KUKA KRL program: EPS_2_25252_DC1_A_20250910061712.src

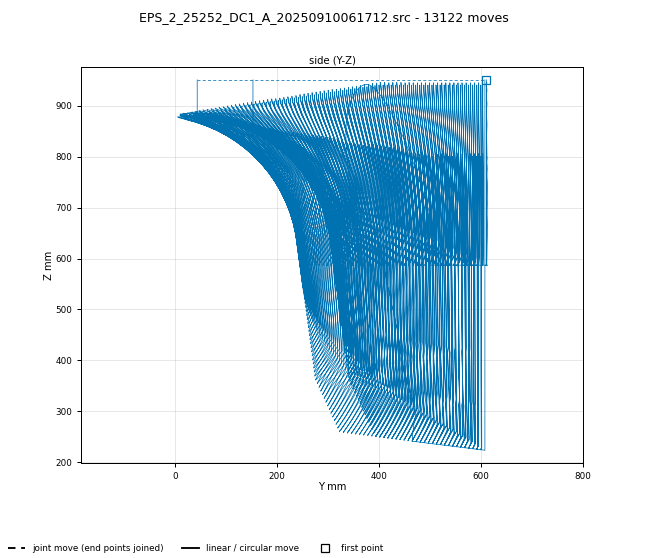
[picture p0: tool path of EPS_2_25252_DC1_A_20250910061712.src, 13122 of 13124 moves have a stored position in this frame; points joined in program order, loops and branches not executed]
&ACCESS RVP
&REL 4
&COMMENT QRS 19112012
&PARAM EDITMASK = *
DEF PART()
EXT BAS (BAS_COMMAND :IN,REAL :IN )
INT I
BAS (#INITMOV,0 )

;KUKA QRS Post kuka4.cps  Date:22-06-2017 !

File_ID=2828

QRS_PRE_INIT()

;Init var - Until changes are made in qrs_pre_init
Outlet_Square_prg=0
Inlet_1_Square_prg=0
Inlet_2_Square_prg=0
Inlet_3_Square_prg=0
Inlet_4_Square_prg=0
Inlet_5_Square_prg=0

Outlet_1={X 0.000, Y 400.000, Z 636.000, B 0.000, E1 0.000 }
Inlet_1={X 0.000, Y 504.550, Z 618.000, B 0.000, E1 206.000 }
Outlet_1_type=610
Inlet_1_type=366
;QRS#1=Sidecore dimensions
;QRS#2=600-24" Concrete
;QRS#3=375-15" PVC SDR 35
;QRS#4=
;QRS#5=
;QRS#6=
;QRS#7=
;QRS#8=
;QRS#9=S306-34L
;QRS#10=20Y PSX
;QRS#11=
;QRS#12=
;QRS#13=
;QRS#14=
;QRS#15=
;QRS#16=1220x127x1295 4,25'
;QRS#17=EPS Height
;QRS#18=941
;QRS#19=*
;QRS#20= UPDATED VERSION 22-06-2017
;QRS#21=*
Outlet_Square=0450
Inlet_1_Square=0250
Inlet_2_Square=0
Inlet_3_Square=0
Inlet_4_Square=0
Inlet_5_Square=0
Mill_Square=1
Outlet_Square_Prg=264
Inlet_1_Square_prg=252

QRS_INIT()

$ADVANCE=5

; T1
PTP {E1 178.399,E2 178.399}
PTP {X 0,Y 610.766,A -85,B 0,C 180,E1 178.399,E2 178.399,E3 0,E4 0,E5 0,E6 0}
QRS_SPEED_INIT()
LIN {X 0,Y 610.766,Z 951,A -85,B 0,C 180,E1 178.399,E2 178.399,E3 0,E4 0,E5 0,E6 0} C_VEL
LIN {X 0,Y 610.766,Z 588.94,A -85,B 0,C 180,E1 178.399,E2 178.399} C_VEL
LIN {X 0,Y 610.795,Z 586.94,A -85,B 0,C 180,E1 178.587,E2 178.587} C_VEL
LIN {X 0,Y 611.848,Z 586.94,A -85,B 0,C 180,E1 181.168,E2 181.168} C_VEL
LIN {X 0,Y 611.871,Z 586.94,A -85,B 0,C 180,E1 188.197,E2 188.197} C_VEL
LIN {X 0,Y 611.797,Z 586.94,A -85,B 0,C 180,E1 195.355,E2 195.355} C_VEL
LIN {X 0,Y 611.804,Z 586.94,A -85,B 0,C 180,E1 202.768,E2 202.768} C_VEL
LIN {X 0,Y 611.794,Z 586.94,A -85,B 0,C 180,E1 210.612,E2 210.612} C_VEL
LIN {X 0,Y 610.594,Z 586.94,A -85,B 0,C 180,E1 217.256,E2 217.256} C_VEL
LIN {X 0,Y 611.723,Z 586.94,A -85,B 0,C 180,E1 219.161,E2 219.161} C_VEL
LIN {X 0,Y 610.308,Z 586.94,A -85,B 0,C 180,E1 222.361,E2 222.361} C_VEL
LIN {X 0,Y 610.612,Z 586.94,A -85,B 0,C 180,E1 225.585,E2 225.585} C_VEL
LIN {X 0,Y 611.691,Z 586.94,A -85,B 0,C 180,E1 227.756,E2 227.756} C_VEL
LIN {X 0,Y 611.857,Z 586.94,A -85,B 0,C 180,E1 235.863,E2 235.863} C_VEL
LIN {X 0,Y 611.311,Z 586.94,A -85,B 0,C 180,E1 236.023,E2 236.023} C_VEL
LIN {X 0,Y 610.597,Z 586.94,A -85,B 0,C 180,E1 236.106,E2 236.106} C_VEL
LIN {X 0,Y 611.51,Z 647.546,A -85,B 0,C 180,E1 237.003,E2 237.003} C_VEL
LIN {X 0,Y 611.588,Z 668.499,A -85,B 0,C 180,E1 237.345,E2 237.345} C_VEL
LIN {X 0,Y 611.321,Z 684.266,A -85,B 0,C 180,E1 237.679,E2 237.679} C_VEL
LIN {X 0,Y 611.684,Z 698.104,A -85,B 0,C 180,E1 238.076,E2 238.076} C_VEL
LIN {X 0,Y 611.753,Z 713.122,A -85,B 0,C 180,E1 238.567,E2 238.567} C_VEL
LIN {X 0,Y 611.745,Z 728.257,A -85,B 0,C 180,E1 239.142,E2 239.142} C_VEL
LIN {X 0,Y 611.602,Z 742.813,A -85,B 0,C 180,E1 239.768,E2 239.768} C_VEL
LIN {X 0,Y 611.469,Z 748.567,A -85,B 0,C 180,E1 240.04,E2 240.04} C_VEL
LIN {X 0,Y 611.62,Z 757.431,A -85,B 0,C 180,E1 240.492,E2 240.492} C_VEL
LIN {X 0,Y 611.575,Z 770.08,A -85,B 0,C 180,E1 241.183,E2 241.183} C_VEL
LIN {X 0,Y 611.546,Z 782.628,A -85,B 0,C 180,E1 241.939,E2 241.939} C_VEL
LIN {X 0,Y 611.656,Z 796.717,A -85,B 0,C 180,E1 242.887,E2 242.887} C_VEL
LIN {X 0,Y 611.627,Z 808.354,A -85,B 0,C 180,E1 243.735,E2 243.735} C_VEL
LIN {X 0,Y 611.516,Z 820.103,A -85,B 0,C 180,E1 244.663,E2 244.663} C_VEL
LIN {X 0,Y 611.31,Z 832.04,A -85,B 0,C 180,E1 245.688,E2 245.688} C_VEL
LIN {X 0,Y 611.351,Z 842.488,A -85,B 0,C 180,E1 246.67,E2 246.67} C_VEL
LIN {X 0,Y 611.614,Z 852.795,A -85,B 0,C 180,E1 247.727,E2 247.727} C_VEL
LIN {X 0,Y 611.705,Z 861.779,A -85,B 0,C 180,E1 248.711,E2 248.711} C_VEL
LIN {X 0,Y 611.244,Z 871.74,A -85,B 0,C 180,E1 249.877,E2 249.877} C_VEL
LIN {X 0,Y 610.937,Z 881.3,A -85,B 0,C 180,E1 251.106,E2 251.106} C_VEL
LIN {X 0,Y 611.042,Z 888.988,A -85,B 0,C 180,E1 252.187,E2 252.187} C_VEL
LIN {X 0,Y 611.571,Z 897.667,A -85,B 0,C 180,E1 253.54,E2 253.54} C_VEL
LIN {X 0,Y 611.79,Z 901.959,A -85,B 0,C 180,E1 254.266,E2 254.266} C_VEL
LIN {X 0,Y 611.426,Z 906.652,A -85,B 0,C 180,E1 255.084,E2 255.084} C_VEL
LIN {X 0,Y 610.99,Z 912.543,A -85,B 0,C 180,E1 256.19,E2 256.19} C_VEL
LIN {X 0,Y 610.849,Z 918.046,A -85,B 0,C 180,E1 257.331,E2 257.331} C_VEL
LIN {X 0,Y 611.295,Z 924.36,A -85,B 0,C 180,E1 258.833,E2 258.833} C_VEL
LIN {X 0,Y 611.852,Z 928.798,A -85,B 0,C 180,E1 260.03,E2 260.03} C_VEL
LIN {X 0,Y 611.223,Z 932.641,A -85,B 0,C 180,E1 261.204,E2 261.204} C_VEL
LIN {X 0,Y 610.765,Z 935.979,A -85,B 0,C 180,E1 262.378,E2 262.378} C_VEL
LIN {X 0,Y 610.652,Z 937.542,A -85,B 0,C 180,E1 262.966,E2 262.966} C_VEL
LIN {X 0,Y 610.835,Z 940.117,A -85,B 0,C 180,E1 264.145,E2 264.145} C_VEL
LIN {X 0,Y 611.39,Z 942.182,A -85,B 0,C 180,E1 265.323,E2 265.323} C_VEL
LIN {X 0,Y 611.706,Z 943.787,A -85,B 0,C 180,E1 266.495,E2 266.495} C_VEL
LIN {X 0,Y 610.903,Z 945.157,A -85,B 0,C 180,E1 267.895,E2 267.895} C_VEL
LIN {X 0,Y 610.566,Z 945.724,A -85,B 0,C 180,E1 268.829,E2 268.829} C_VEL
LIN {X 0,Y 610.611,Z 945.959,A -85,B 0,C 180,E1 270.175,E2 270.175} C_VEL
LIN {X 0,Y 611.002,Z 945.713,A -85,B 0,C 180,E1 271.168,E2 271.168} C_VEL
LIN {X 0,Y 611.64,Z 945.019,A -85,B 0,C 180,E1 272.253,E2 272.253} C_VEL
LIN {X 0,Y 611.557,Z 944.17,A -85,B 0,C 180,E1 273.193,E2 273.193} C_VEL
LIN {X 0,Y 610.851,Z 942.2,A -85,B 0,C 180,E1 274.679,E2 274.679} C_VEL
LIN {X 0,Y 610.654,Z 940.123,A -85,B 0,C 180,E1 275.855,E2 275.855} C_VEL
LIN {X 0,Y 610.92,Z 937.546,A -85,B 0,C 180,E1 277.029,E2 277.029} C_VEL
LIN {X 0,Y 611.534,Z 934.39,A -85,B 0,C 180,E1 278.199,E2 278.199} C_VEL
LIN {X 0,Y 611.853,Z 932.642,A -85,B 0,C 180,E1 278.785,E2 278.785} C_VEL
LIN {X 0,Y 611.268,Z 928.807,A -85,B 0,C 180,E1 279.977,E2 279.977} C_VEL
LIN {X 0,Y 610.798,Z 923.162,A -85,B 0,C 180,E1 281.472,E2 281.472} C_VEL
LIN {X 0,Y 610.882,Z 918.056,A -85,B 0,C 180,E1 282.666,E2 282.666} C_VEL
LIN {X 0,Y 611.577,Z 910.301,A -85,B 0,C 180,E1 284.234,E2 284.234} C_VEL
LIN {X 0,Y 611.794,Z 906.723,A -85,B 0,C 180,E1 284.894,E2 284.894} C_VEL
LIN {X 0,Y 611.436,Z 902.319,A -85,B 0,C 180,E1 285.683,E2 285.683} C_VEL
LIN {X 0,Y 611.057,Z 897.089,A -85,B 0,C 180,E1 286.572,E2 286.572} C_VEL
LIN {X 0,Y 610.862,Z 887.941,A -85,B 0,C 180,E1 287.97,E2 287.97} C_VEL
LIN {X 0,Y 611.214,Z 879.031,A -85,B 0,C 180,E1 289.192,E2 289.192} C_VEL
LIN {X 0,Y 611.72,Z 869.206,A -85,B 0,C 180,E1 290.415,E2 290.415} C_VEL
LIN {X 0,Y 611.518,Z 859.844,A -85,B 0,C 180,E1 291.512,E2 291.512} C_VEL
LIN {X 0,Y 611.23,Z 849.887,A -85,B 0,C 180,E1 292.592,E2 292.592} C_VEL
LIN {X 0,Y 611.217,Z 839.652,A -85,B 0,C 180,E1 293.61,E2 293.61} C_VEL
LIN {X 0,Y 611.473,Z 828.289,A -85,B 0,C 180,E1 294.639,E2 294.639} C_VEL
LIN {X 0,Y 611.646,Z 817.642,A -85,B 0,C 180,E1 295.534,E2 295.534} C_VEL
LIN {X 0,Y 611.637,Z 805.784,A -85,B 0,C 180,E1 296.46,E2 296.46} C_VEL
LIN {X 0,Y 611.539,Z 793.169,A -85,B 0,C 180,E1 297.366,E2 297.366} C_VEL
LIN {X 0,Y 611.545,Z 780.808,A -85,B 0,C 180,E1 298.176,E2 298.176} C_VEL
LIN {X 0,Y 611.615,Z 766.332,A -85,B 0,C 180,E1 299.027,E2 299.027} C_VEL
LIN {X 0,Y 611.558,Z 756.226,A -85,B 0,C 180,E1 299.577,E2 299.577} C_VEL
LIN {X 0,Y 611.728,Z 739.176,A -85,B 0,C 180,E1 300.392,E2 300.392} C_VEL
LIN {X 0,Y 611.714,Z 723.993,A -85,B 0,C 180,E1 301.03,E2 301.03} C_VEL
LIN {X 0,Y 611.675,Z 709.715,A -85,B 0,C 180,E1 301.554,E2 301.554} C_VEL
LIN {X 0,Y 611.325,Z 695.349,A -85,B 0,C 180,E1 302.025,E2 302.025} C_VEL
LIN {X 0,Y 611.698,Z 679.814,A -85,B 0,C 180,E1 302.406,E2 302.406} C_VEL
LIN {X 0,Y 611.757,Z 665.783,A -85,B 0,C 180,E1 302.698,E2 302.698} C_VEL
LIN {X 0,Y 611.651,Z 645.532,A -85,B 0,C 180,E1 303.016,E2 303.016} C_VEL
LIN {X 0,Y 610.854,Z 596.983,A -85,B 0,C 180,E1 303.735,E2 303.735} C_VEL
LIN {X 0,Y 610.662,Z 586.94,A -85,B 0,C 180,E1 303.893,E2 303.893} C_VEL
LIN {X 0,Y 611.322,Z 586.94,A -85,B 0,C 180,E1 303.972,E2 303.972} C_VEL
LIN {X 0,Y 611.676,Z 586.94,A -85,B 0,C 180,E1 304.64,E2 304.64} C_VEL
LIN {X 0,Y 611.825,Z 586.94,A -85,B 0,C 180,E1 309.151,E2 309.151} C_VEL
LIN {X 0,Y 610.37,Z 586.94,A -85,B 0,C 180,E1 312.353,E2 312.353} C_VEL
LIN {X 0,Y 610.667,Z 586.94,A -85,B 0,C 180,E1 315.577,E2 315.577} C_VEL
LIN {X 0,Y 611.742,Z 586.94,A -85,B 0,C 180,E1 317.761,E2 317.761} C_VEL
LIN {X 0,Y 610.224,Z 586.94,A -85,B 0,C 180,E1 323.686,E2 323.686} C_VEL
LIN {X 0,Y 611.725,Z 586.94,A -85,B 0,C 180,E1 326.634,E2 326.634} C_VEL
LIN {X 0,Y 611.738,Z 586.94,A -85,B 0,C 180,E1 334.673,E2 334.673} C_VEL
LIN {X 0,Y 611.49,Z 586.94,A -85,B 0,C 180,E1 343.289,E2 343.289} C_VEL
LIN {X 0,Y 611.249,Z 586.94,A -85,B 0,C 180,E1 344.631,E2 344.631} C_VEL
LIN {X 0,Y 611.788,Z 586.94,A -85,B 0,C 180,E1 351.802,E2 351.802} C_VEL
LIN {X 0,Y 611.834,Z 586.94,A -85,B 0,C 180,E1 358.832,E2 358.832} C_VEL
LIN {X 0,Y 611.791,Z 586.94,A -85,B 0,C 180,E1 365.845,E2 365.845} C_VEL
LIN {X 0,Y 611.835,Z 586.94,A -85,B 0,C 180,E1 372.946,E2 372.946} C_VEL
LIN {X 0,Y 611.779,Z 586.94,A -85,B 0,C 180,E1 380.259,E2 380.259} C_VEL
LIN {X 0,Y 611.755,Z 586.94,A -85,B 0,C 180,E1 387.936,E2 387.936} C_VEL
LIN {X 0,Y 610.34,Z 586.94,A -85,B 0,C 180,E1 393.168,E2 393.168} C_VEL
LIN {X 0,Y 611.785,Z 586.94,A -85,B 0,C 180,E1 396.205,E2 396.205} C_VEL
LIN {X 0,Y 611.323,Z 586.94,A -85,B 0,C 180,E1 397.349,E2 397.349} C_VEL
LIN {X 0,Y 611.836,Z 586.94,A -85,B 0,C 180,E1 403.144,E2 403.144} C_VEL
LIN {X 0,Y 611.437,Z 586.94,A -85,B 0,C 180,E1 403.288,E2 403.288} C_VEL
LIN {X 0,Y 611.426,Z 596.264,A -85,B 0,C 180,E1 403.448,E2 403.448} C_VEL
LIN {X 0,Y 611.785,Z 623.475,A -85,B 0,C 180,E1 403.804,E2 403.804} C_VEL
LIN {X 0,Y 611.801,Z 632.118,A -85,B 0,C 180,E1 403.947,E2 403.947} C_VEL
LIN {X 0,Y 611.734,Z 641.309,A -85,B 0,C 180,E1 404.136,E2 404.136} C_VEL
LIN {X 0,Y 611.726,Z 648.588,A -85,B 0,C 180,E1 404.316,E2 404.316} C_VEL
LIN {X 0,Y 611.81,Z 658.939,A -85,B 0,C 180,E1 404.626,E2 404.626} C_VEL
LIN {X 0,Y 611.799,Z 668.311,A -85,B 0,C 180,E1 404.953,E2 404.953} C_VEL
LIN {X 0,Y 611.811,Z 677.548,A -85,B 0,C 180,E1 405.323,E2 405.323} C_VEL
LIN {X 0,Y 611.792,Z 686.258,A -85,B 0,C 180,E1 405.718,E2 405.718} C_VEL
LIN {X 0,Y 611.755,Z 693.578,A -85,B 0,C 180,E1 406.083,E2 406.083} C_VEL
LIN {X 0,Y 611.679,Z 703.091,A -85,B 0,C 180,E1 406.614,E2 406.614} C_VEL
LIN {X 0,Y 611.54,Z 712.053,A -85,B 0,C 180,E1 407.172,E2 407.172} C_VEL
LIN {X 0,Y 611.518,Z 719.064,A -85,B 0,C 180,E1 407.653,E2 407.653} C_VEL
LIN {X 0,Y 611.656,Z 726.904,A -85,B 0,C 180,E1 408.246,E2 408.246} C_VEL
LIN {X 0,Y 611.808,Z 734.808,A -85,B 0,C 180,E1 408.903,E2 408.903} C_VEL
LIN {X 0,Y 611.752,Z 740.864,A -85,B 0,C 180,E1 409.445,E2 409.445} C_VEL
LIN {X 0,Y 611.519,Z 747.37,A -85,B 0,C 180,E1 410.073,E2 410.073} C_VEL
LIN {X 0,Y 611.286,Z 754.307,A -85,B 0,C 180,E1 410.808,E2 410.808} C_VEL
LIN {X 0,Y 611.275,Z 759.983,A -85,B 0,C 180,E1 411.467,E2 411.467} C_VEL
LIN {X 0,Y 611.474,Z 765.259,A -85,B 0,C 180,E1 412.136,E2 412.136} C_VEL
LIN {X 0,Y 611.815,Z 771.733,A -85,B 0,C 180,E1 413.047,E2 413.047} C_VEL
LIN {X 0,Y 611.775,Z 774.744,A -85,B 0,C 180,E1 413.495,E2 413.495} C_VEL
LIN {X 0,Y 611.312,Z 780.353,A -85,B 0,C 180,E1 414.417,E2 414.417} C_VEL
LIN {X 0,Y 611.03,Z 784.515,A -85,B 0,C 180,E1 415.18,E2 415.18} C_VEL
LIN {X 0,Y 611.072,Z 789.541,A -85,B 0,C 180,E1 416.243,E2 416.243} C_VEL
LIN {X 0,Y 611.399,Z 792.933,A -85,B 0,C 180,E1 417.064,E2 417.064} C_VEL
LIN {X 0,Y 611.88,Z 796.656,A -85,B 0,C 180,E1 418.124,E2 418.124} C_VEL
LIN {X 0,Y 611.543,Z 798.59,A -85,B 0,C 180,E1 418.743,E2 418.743} C_VEL
LIN {X 0,Y 611.002,Z 801.321,A -85,B 0,C 180,E1 419.81,E2 419.81} C_VEL
LIN {X 0,Y 610.85,Z 802.311,A -85,B 0,C 180,E1 420.263,E2 420.263} C_VEL
LIN {X 0,Y 610.888,Z 804.098,A -85,B 0,C 180,E1 421.298,E2 421.298} C_VEL
LIN {X 0,Y 611.19,Z 804.968,A -85,B 0,C 180,E1 422.036,E2 422.036} C_VEL
LIN {X 0,Y 611.725,Z 805.707,A -85,B 0,C 180,E1 423.014,E2 423.014} C_VEL
LIN {X 0,Y 611.599,Z 805.938,A -85,B 0,C 180,E1 423.841,E2 423.841} C_VEL
LIN {X 0,Y 611.17,Z 805.82,A -85,B 0,C 180,E1 424.65,E2 424.65} C_VEL
LIN {X 0,Y 610.885,Z 805.27,A -85,B 0,C 180,E1 425.565,E2 425.565} C_VEL
LIN {X 0,Y 610.97,Z 804.103,A -85,B 0,C 180,E1 426.607,E2 426.607} C_VEL
LIN {X 0,Y 611.606,Z 801.736,A -85,B 0,C 180,E1 427.897,E2 427.897} C_VEL
LIN {X 0,Y 611.834,Z 800.373,A -85,B 0,C 180,E1 428.496,E2 428.496} C_VEL
LIN {X 0,Y 611.547,Z 798.741,A -85,B 0,C 180,E1 429.111,E2 429.111} C_VEL
LIN {X 0,Y 611.047,Z 794.846,A -85,B 0,C 180,E1 430.338,E2 430.338} C_VEL
LIN {X 0,Y 611.021,Z 791.266,A -85,B 0,C 180,E1 431.265,E2 431.265} C_VEL
LIN {X 0,Y 611.188,Z 788.592,A -85,B 0,C 180,E1 431.886,E2 431.886} C_VEL
LIN {X 0,Y 611.695,Z 783.499,A -85,B 0,C 180,E1 432.91,E2 432.91} C_VEL
LIN {X 0,Y 611.796,Z 780.157,A -85,B 0,C 180,E1 433.522,E2 433.522} C_VEL
LIN {X 0,Y 611.433,Z 774.547,A -85,B 0,C 180,E1 434.45,E2 434.45} C_VEL
LIN {X 0,Y 611.223,Z 769.16,A -85,B 0,C 180,E1 435.249,E2 435.249} C_VEL
LIN {X 0,Y 611.303,Z 762.983,A -85,B 0,C 180,E1 436.07,E2 436.07} C_VEL
LIN {X 0,Y 611.603,Z 756.399,A -85,B 0,C 180,E1 436.858,E2 436.858} C_VEL
LIN {X 0,Y 611.811,Z 750.518,A -85,B 0,C 180,E1 437.503,E2 437.503} C_VEL
LIN {X 0,Y 611.744,Z 744.701,A -85,B 0,C 180,E1 438.099,E2 438.099} C_VEL
LIN {X 0,Y 611.517,Z 736.799,A -85,B 0,C 180,E1 438.839,E2 438.839} C_VEL
LIN {X 0,Y 611.419,Z 729.861,A -85,B 0,C 180,E1 439.432,E2 439.432} C_VEL
LIN {X 0,Y 611.525,Z 722.186,A -85,B 0,C 180,E1 440.027,E2 440.027} C_VEL
LIN {X 0,Y 611.691,Z 714.816,A -85,B 0,C 180,E1 440.548,E2 440.548} C_VEL
LIN {X 0,Y 611.77,Z 706.806,A -85,B 0,C 180,E1 441.066,E2 441.066} C_VEL
LIN {X 0,Y 611.815,Z 697.975,A -85,B 0,C 180,E1 441.583,E2 441.583} C_VEL
LIN {X 0,Y 611.708,Z 689.71,A -85,B 0,C 180,E1 442.024,E2 442.024} C_VEL
LIN {X 0,Y 611.662,Z 682.082,A -85,B 0,C 180,E1 442.391,E2 442.391} C_VEL
LIN {X 0,Y 611.694,Z 673.493,A -85,B 0,C 180,E1 442.76,E2 442.76} C_VEL
LIN {X 0,Y 611.796,Z 663.564,A -85,B 0,C 180,E1 443.128,E2 443.128} C_VEL
LIN {X 0,Y 611.657,Z 654.069,A -85,B 0,C 180,E1 443.439,E2 443.439} C_VEL
LIN {X 0,Y 611.841,Z 644.324,A -85,B 0,C 180,E1 443.698,E2 443.698} C_VEL
LIN {X 0,Y 611.835,Z 635.38,A -85,B 0,C 180,E1 443.9,E2 443.9} C_VEL
LIN {X 0,Y 611.824,Z 626.266,A -85,B 0,C 180,E1 444.064,E2 444.064} C_VEL
LIN {X 0,Y 611.79,Z 606.948,A -85,B 0,C 180,E1 444.318,E2 444.318} C_VEL
LIN {X 0,Y 611.528,Z 586.94,A -85,B 0,C 180,E1 444.573,E2 444.573} C_VEL
LIN {X 0,Y 611.869,Z 586.94,A -85,B 0,C 180,E1 444.752,E2 444.752} C_VEL
LIN {X 0,Y 611.873,Z 586.94,A -85,B 0,C 180,E1 451.168,E2 451.168} C_VEL
LIN {X 0,Y 611.821,Z 586.94,A -85,B 0,C 180,E1 458.198,E2 458.198} C_VEL
LIN {X 0,Y 611.842,Z 586.94,A -85,B 0,C 180,E1 465.354,E2 465.354} C_VEL
LIN {X 0,Y 611.828,Z 586.94,A -85,B 0,C 180,E1 472.768,E2 472.768} C_VEL
LIN {X 0,Y 611.808,Z 586.94,A -85,B 0,C 180,E1 480.611,E2 480.611} C_VEL
LIN {X 0,Y 610.644,Z 586.94,A -85,B 0,C 180,E1 487.264,E2 487.264} C_VEL
LIN {X 0,Y 611.777,Z 586.94,A -85,B 0,C 180,E1 489.157,E2 489.157} C_VEL
LIN {X 0,Y 610.366,Z 586.94,A -85,B 0,C 180,E1 492.357,E2 492.357} C_VEL
LIN {X 0,Y 610.675,Z 586.94,A -85,B 0,C 180,E1 495.579,E2 495.579} C_VEL
LIN {X 0,Y 611.764,Z 586.94,A -85,B 0,C 180,E1 497.765,E2 497.765} C_VEL
LIN {X 0,Y 610.281,Z 586.94,A -85,B 0,C 180,E1 503.691,E2 503.691} C_VEL
LIN {X 0,Y 611.799,Z 586.94,A -85,B 0,C 180,E1 506.638,E2 506.638} C_VEL
LIN {X 0,Y 611.815,Z 586.94,A -85,B 0,C 180,E1 514.678,E2 514.678} C_VEL
LIN {X 0,Y 611.539,Z 586.94,A -85,B 0,C 180,E1 523.281,E2 523.281} C_VEL
LIN {X 0,Y 611.682,Z 586.94,A -85,B 0,C 180,E1 524.643,E2 524.643} C_VEL
LIN {X 0,Y 611.854,Z 586.94,A -85,B 0,C 180,E1 527.055,E2 527.055} C_VEL
LIN {X 0,Y 611.855,Z 586.94,A -85,B 0,C 180,E1 534.156,E2 534.156} C_VEL
LIN {X 0,Y 610.795,Z 586.94,A -85,B 0,C 180,E1 538.587,E2 538.587} C_VEL
LIN {X 0,Y 603.322,Z 586.94,A -85,B 0,C 180,E1 541.885,E2 541.885} C_VEL
LIN {X 0,Y 603.193,Z 586.94,A -85,B 0,C 180,E1 549.38,E2 549.38} C_VEL
LIN {X 0,Y 603.019,Z 586.94,A -85,B 0,C 180,E1 556.787,E2 556.787} C_VEL
LIN {X 0,Y 602.84,Z 586.94,A -85,B 0,C 180,E1 564.501,E2 564.501} C_VEL
LIN {X 0,Y 602.62,Z 586.94,A -85,B 0,C 180,E1 572.477,E2 572.477} C_VEL
LIN {X 0,Y 603.236,Z 586.94,A -85,B 0,C 180,E1 579.89,E2 579.89} C_VEL
LIN {X 0,Y 603.395,Z 586.94,A -85,B 0,C 180,E1 588.204,E2 588.204} C_VEL
LIN {X 0,Y 603.949,Z 588.901,A -85,B 0,C 180,E1 595.713,E2 595.713} C_VEL
LIN {X 0,Y 604.773,Z 695.526,A -85,B 0,C 180,E1 597.59,E2 597.59} C_VEL
LIN {X 0,Y 604.454,Z 760.206,A -85,B 0,C 180,E1 600.259,E2 600.259} C_VEL
LIN {X 0,Y 604.022,Z 820.002,A -85,B 0,C 180,E1 604.317,E2 604.317} C_VEL
LIN {X 0,Y 603.53,Z 871.532,A -85,B 0,C 180,E1 609.581,E2 609.581} C_VEL
LIN {X 0,Y 603.283,Z 909.881,A -85,B 0,C 180,E1 615.486,E2 615.486} C_VEL
LIN {X 0,Y 603.167,Z 933.377,A -85,B 0,C 180,E1 621.317,E2 621.317} C_VEL
LIN {X 0,Y 603.668,Z 943.765,A -85,B 0,C 180,E1 626.396,E2 626.396} C_VEL
LIN {X 0,Y 603.583,Z 945.149,A -85,B 0,C 180,E1 632.161,E2 632.161} C_VEL
LIN {X 0,Y 603.804,Z 933.381,A -85,B 0,C 180,E1 638.672,E2 638.672} C_VEL
LIN {X 0,Y 603.711,Z 905.639,A -85,B 0,C 180,E1 645.303,E2 645.303} C_VEL
LIN {X 0,Y 603.811,Z 865.155,A -85,B 0,C 180,E1 651.178,E2 651.178} C_VEL
LIN {X 0,Y 604.16,Z 813.982,A -85,B 0,C 180,E1 656.166,E2 656.166} C_VEL
LIN {X 0,Y 604.519,Z 753.653,A -85,B 0,C 180,E1 660.091,E2 660.091} C_VEL
LIN {X 0,Y 604.745,Z 687.82,A -85,B 0,C 180,E1 662.62,E2 662.62} C_VEL
LIN {X 0,Y 603.579,Z 586.94,A -85,B 0,C 180,E1 664.45,E2 664.45} C_VEL
LIN {X 0,Y 602.435,Z 586.94,A -85,B 0,C 180,E1 672.07,E2 672.07} C_VEL
LIN {X 0,Y 603.35,Z 586.94,A -85,B 0,C 180,E1 678.259,E2 678.259} C_VEL
LIN {X 0,Y 603.179,Z 586.94,A -85,B 0,C 180,E1 687.437,E2 687.437} C_VEL
LIN {X 0,Y 603.092,Z 586.94,A -85,B 0,C 180,E1 695.51,E2 695.51} C_VEL
LIN {X 0,Y 603.188,Z 586.94,A -85,B 0,C 180,E1 704.718,E2 704.718} C_VEL
LIN {X 0,Y 602.84,Z 586.94,A -85,B 0,C 180,E1 713.887,E2 713.887} C_VEL
LIN {X 0,Y 602.921,Z 586.94,A -85,B 0,C 180,E1 720.748,E2 720.748} C_VEL
LIN {X 0,Y 602.822,Z 586.94,A -85,B 0,C 180,E1 727.983,E2 727.983} C_VEL
LIN {X 0,Y 602.745,Z 586.94,A -85,B 0,C 180,E1 735.351,E2 735.351} C_VEL
LIN {X 0,Y 603.092,Z 586.94,A -85,B 0,C 180,E1 741.419,E2 741.419} C_VEL
LIN {X 0,Y 602.704,Z 586.94,A -85,B 0,C 180,E1 749.698,E2 749.698} C_VEL
LIN {X 0,Y 603.072,Z 586.94,A -85,B 0,C 180,E1 758.078,E2 758.078} C_VEL
LIN {X 0,Y 603.811,Z 587.895,A -85,B 0,C 180,E1 763.073,E2 763.073} C_VEL
LIN {X 0,Y 604.249,Z 657.832,A -85,B 0,C 180,E1 764.337,E2 764.337} C_VEL
LIN {X 0,Y 603.872,Z 709.067,A -85,B 0,C 180,E1 766.753,E2 766.753} C_VEL
LIN {X 0,Y 603.464,Z 752.858,A -85,B 0,C 180,E1 770.467,E2 770.467} C_VEL
LIN {X 0,Y 603.152,Z 783.489,A -85,B 0,C 180,E1 774.87,E2 774.87} C_VEL
LIN {X 0,Y 603.032,Z 801.266,A -85,B 0,C 180,E1 779.726,E2 779.726} C_VEL
LIN {X 0,Y 603.557,Z 805.994,A -85,B 0,C 180,E1 783.897,E2 783.897} C_VEL
LIN {X 0,Y 603.6,Z 799.212,A -85,B 0,C 180,E1 789.007,E2 789.007} C_VEL
LIN {X 0,Y 603.604,Z 777.311,A -85,B 0,C 180,E1 794.134,E2 794.134} C_VEL
LIN {X 0,Y 603.763,Z 741.658,A -85,B 0,C 180,E1 798.585,E2 798.585} C_VEL
LIN {X 0,Y 604.092,Z 695.259,A -85,B 0,C 180,E1 801.968,E2 801.968} C_VEL
LIN {X 0,Y 604.312,Z 643.902,A -85,B 0,C 180,E1 803.965,E2 803.965} C_VEL
LIN {X 0,Y 603.752,Z 586.94,A -85,B 0,C 180,E1 804.954,E2 804.954} C_VEL
LIN {X 0,Y 603.31,Z 586.94,A -85,B 0,C 180,E1 812.163,E2 812.163} C_VEL
LIN {X 0,Y 603.178,Z 586.94,A -85,B 0,C 180,E1 819.413,E2 819.413} C_VEL
LIN {X 0,Y 603.039,Z 586.94,A -85,B 0,C 180,E1 826.822,E2 826.822} C_VEL
LIN {X 0,Y 602.827,Z 586.94,A -85,B 0,C 180,E1 834.543,E2 834.543} C_VEL
LIN {X 0,Y 602.667,Z 586.94,A -85,B 0,C 180,E1 842.47,E2 842.47} C_VEL
LIN {X 0,Y 603.277,Z 586.94,A -85,B 0,C 180,E1 849.9,E2 849.9} C_VEL
LIN {X 0,Y 603.426,Z 586.94,A -85,B 0,C 180,E1 858.191,E2 858.191} C_VEL
LIN {X 0,Y 603.266,Z 586.94,A -85,B 0,C 180,E1 867.427,E2 867.427} C_VEL
LIN {X 0,Y 603.207,Z 586.94,A -85,B 0,C 180,E1 875.455,E2 875.455} C_VEL
LIN {X 0,Y 603.643,Z 586.94,A -85,B 0,C 180,E1 885.438,E2 885.438} C_VEL
LIN {X 0,Y 603.401,Z 586.94,A -85,B 0,C 180,E1 894.925,E2 894.925} C_VEL
LIN {X 0,Y 603.322,Z 586.94,A -85,B 0,C 180,E1 901.885,E2 901.885} C_VEL
LIN {X 0,Y 594.758,Z 586.94,A -85,B 0,C 180,E1 905.177,E2 905.177} C_VEL
LIN {X 0,Y 594.724,Z 586.94,A -85,B 0,C 180,E1 911,E2 911} C_VEL
LIN {X 0,Y 594.921,Z 586.94,A -85,B 0,C 180,E1 917.022,E2 917.022} C_VEL
LIN {X 0,Y 594.638,Z 586.94,A -85,B 0,C 180,E1 925.045,E2 925.045} C_VEL
LIN {X 0,Y 595.168,Z 586.94,A -85,B 0,C 180,E1 931.467,E2 931.467} C_VEL
LIN {X 0,Y 594.632,Z 586.94,A -85,B 0,C 180,E1 941.161,E2 941.161} C_VEL
LIN {X 0,Y 594.731,Z 586.94,A -85,B 0,C 180,E1 949.408,E2 949.408} C_VEL
LIN {X 0,Y 595.456,Z 588.194,A -85,B 0,C 180,E1 955.144,E2 955.144} C_VEL
LIN {X 0,Y 597.833,Z 627.641,A -85,B 0,C 180,E1 955.865,E2 955.865} C_VEL
LIN {X 0,Y 597.979,Z 702.266,A -85,B 0,C 180,E1 957.391,E2 957.391} C_VEL
LIN {X 0,Y 597.25,Z 766.884,A -85,B 0,C 180,E1 960.235,E2 960.235} C_VEL
LIN {X 0,Y 596.384,Z 825.898,A -85,B 0,C 180,E1 964.484,E2 964.484} C_VEL
LIN {X 0,Y 595.612,Z 874.486,A -85,B 0,C 180,E1 969.687,E2 969.687} C_VEL
LIN {X 0,Y 595.289,Z 911.334,A -85,B 0,C 180,E1 975.565,E2 975.565} C_VEL
LIN {X 0,Y 595.231,Z 933.377,A -85,B 0,C 180,E1 981.2,E2 981.2} C_VEL
LIN {X 0,Y 595.657,Z 943.765,A -85,B 0,C 180,E1 986.348,E2 986.348} C_VEL
LIN {X 0,Y 595.571,Z 945.149,A -85,B 0,C 180,E1 992.19,E2 992.19} C_VEL
LIN {X 0,Y 595.803,Z 933.381,A -85,B 0,C 180,E1 998.79,E2 998.79} C_VEL
LIN {X 0,Y 595.675,Z 905.64,A -85,B 0,C 180,E1 1005.515,E2 1005.515} C_VEL
LIN {X 0,Y 596.03,Z 865.156,A -85,B 0,C 180,E1 1011.468,E2 1011.468} C_VEL
LIN {X 0,Y 596.699,Z 813.947,A -85,B 0,C 180,E1 1016.521,E2 1016.521} C_VEL
LIN {X 0,Y 597.448,Z 753.657,A -85,B 0,C 180,E1 1020.485,E2 1020.485} C_VEL
LIN {X 0,Y 597.999,Z 687.837,A -85,B 0,C 180,E1 1023.034,E2 1023.034} C_VEL
LIN {X 0,Y 595.842,Z 589.198,A -85,B 0,C 180,E1 1024.816,E2 1024.816} C_VEL
LIN {X 0,Y 595.496,Z 586.94,A -85,B 0,C 180,E1 1024.985,E2 1024.985} C_VEL
LIN {X 0,Y 594.284,Z 586.94,A -85,B 0,C 180,E1 1033.366,E2 1033.366} C_VEL
LIN {X 0,Y 594.638,Z 586.94,A -85,B 0,C 180,E1 1039.457,E2 1039.457} C_VEL
LIN {X 0,Y 594.651,Z 586.94,A -85,B 0,C 180,E1 1048.503,E2 1048.503} C_VEL
LIN {X 0,Y 594.438,Z 586.94,A -85,B 0,C 180,E1 1056.731,E2 1056.731} C_VEL
LIN {X 0,Y 595.2,Z 586.94,A -85,B 0,C 180,E1 1064.507,E2 1064.507} C_VEL
LIN {X 0,Y 594.971,Z 586.94,A -85,B 0,C 180,E1 1073.44,E2 1073.44} C_VEL
LIN {X 0,Y 594.931,Z 586.94,A -85,B 0,C 180,E1 1080.758,E2 1080.758} C_VEL
LIN {X 0,Y 594.794,Z 586.94,A -85,B 0,C 180,E1 1088.091,E2 1088.091} C_VEL
LIN {X 0,Y 594.697,Z 586.94,A -85,B 0,C 180,E1 1095.564,E2 1095.564} C_VEL
LIN {X 0,Y 594.937,Z 586.94,A -85,B 0,C 180,E1 1101.728,E2 1101.728} C_VEL
LIN {X 0,Y 594.663,Z 586.94,A -85,B 0,C 180,E1 1109.862,E2 1109.862} C_VEL
LIN {X 0,Y 595.507,Z 586.94,A -85,B 0,C 180,E1 1116.805,E2 1116.805} C_VEL
LIN {X 0,Y 595.813,Z 588.595,A -85,B 0,C 180,E1 1122.788,E2 1122.788} C_VEL
LIN {X 0,Y 596.668,Z 658.067,A -85,B 0,C 180,E1 1124.085,E2 1124.085} C_VEL
LIN {X 0,Y 596.164,Z 709.072,A -85,B 0,C 180,E1 1126.523,E2 1126.523} C_VEL
LIN {X 0,Y 595.597,Z 752.976,A -85,B 0,C 180,E1 1130.3,E2 1130.3} C_VEL
LIN {X 0,Y 595.232,Z 783.05,A -85,B 0,C 180,E1 1134.665,E2 1134.665} C_VEL
LIN {X 0,Y 595.183,Z 800.668,A -85,B 0,C 180,E1 1139.392,E2 1139.392} C_VEL
LIN {X 0,Y 595.115,Z 805.785,A -85,B 0,C 180,E1 1144.872,E2 1144.872} C_VEL
LIN {X 0,Y 595.237,Z 796.927,A -85,B 0,C 180,E1 1149.869,E2 1149.869} C_VEL
LIN {X 0,Y 595.464,Z 774.734,A -85,B 0,C 180,E1 1154.706,E2 1154.706} C_VEL
LIN {X 0,Y 595.851,Z 738.551,A -85,B 0,C 180,E1 1159.082,E2 1159.082} C_VEL
LIN {X 0,Y 596.391,Z 691.883,A -85,B 0,C 180,E1 1162.394,E2 1162.394} C_VEL
LIN {X 0,Y 596.842,Z 639.005,A -85,B 0,C 180,E1 1164.346,E2 1164.346} C_VEL
LIN {X 0,Y 595.588,Z 586.94,A -85,B 0,C 180,E1 1165.251,E2 1165.251} C_VEL
LIN {X 0,Y 594.807,Z 586.94,A -85,B 0,C 180,E1 1173.658,E2 1173.658} C_VEL
LIN {X 0,Y 594.771,Z 586.94,A -85,B 0,C 180,E1 1180.767,E2 1180.767} C_VEL
LIN {X 0,Y 594.945,Z 586.94,A -85,B 0,C 180,E1 1187.058,E2 1187.058} C_VEL
LIN {X 0,Y 594.663,Z 586.94,A -85,B 0,C 180,E1 1195.035,E2 1195.035} C_VEL
LIN {X 0,Y 595.196,Z 586.94,A -85,B 0,C 180,E1 1201.512,E2 1201.512} C_VEL
LIN {X 0,Y 594.689,Z 586.94,A -85,B 0,C 180,E1 1211.152,E2 1211.152} C_VEL
LIN {X 0,Y 594.704,Z 586.94,A -85,B 0,C 180,E1 1219.389,E2 1219.389} C_VEL
LIN {X 0,Y 594.776,Z 586.94,A -85,B 0,C 180,E1 1228.445,E2 1228.445} C_VEL
LIN {X 0,Y 594.524,Z 586.94,A -85,B 0,C 180,E1 1236.674,E2 1236.674} C_VEL
LIN {X 0,Y 595.679,Z 586.94,A -85,B 0,C 180,E1 1245.971,E2 1245.971} C_VEL
LIN {X 0,Y 595.412,Z 586.94,A -85,B 0,C 180,E1 1254.856,E2 1254.856} C_VEL
LIN {X 0,Y 595.299,Z 586.94,A -85,B 0,C 180,E1 1262.163,E2 1262.163} C_VEL
LIN {X 0,Y 594.758,Z 586.94,A -85,B 0,C 180,E1 1265.177,E2 1265.177} C_VEL
LIN {X 0,Y 587.421,Z 586.94,A -85,B 0,C 180,E1 1268.543,E2 1268.543} C_VEL
LIN {X 0,Y 586.834,Z 586.94,A -85,B 0,C 180,E1 1277.264,E2 1277.264} C_VEL
LIN {X 0,Y 586.586,Z 586.94,A -85,B 0,C 180,E1 1285.226,E2 1285.226} C_VEL
LIN {X 0,Y 586.496,Z 586.94,A -85,B 0,C 180,E1 1292.762,E2 1292.762} C_VEL
LIN {X 0,Y 586.631,Z 586.94,A -85,B 0,C 180,E1 1301.215,E2 1301.215} C_VEL
LIN {X 0,Y 586.638,Z 586.94,A -85,B 0,C 180,E1 1309.668,E2 1309.668} C_VEL
LIN {X 0,Y 587.152,Z 588.322,A -85,B 0,C 180,E1 1314.579,E2 1314.579} C_VEL
LIN {X 0,Y 590.898,Z 602.269,A -85,B 0,C 180,E1 1315.04,E2 1315.04} C_VEL
LIN {X 0,Y 591.171,Z 697.397,A -85,B 0,C 180,E1 1316.805,E2 1316.805} C_VEL
LIN {X 0,Y 590.176,Z 763.009,A -85,B 0,C 180,E1 1319.622,E2 1319.622} C_VEL
LIN {X 0,Y 589.051,Z 821.97,A -85,B 0,C 180,E1 1323.791,E2 1323.791} C_VEL
LIN {X 0,Y 588.087,Z 871.535,A -85,B 0,C 180,E1 1329.02,E2 1329.02} C_VEL
LIN {X 0,Y 587.472,Z 910.819,A -85,B 0,C 180,E1 1335.268,E2 1335.268} C_VEL
LIN {X 0,Y 587.317,Z 933.376,A -85,B 0,C 180,E1 1341.081,E2 1341.081} C_VEL
LIN {X 0,Y 587.636,Z 943.765,A -85,B 0,C 180,E1 1346.298,E2 1346.298} C_VEL
LIN {X 0,Y 587.56,Z 945.149,A -85,B 0,C 180,E1 1352.22,E2 1352.22} C_VEL
LIN {X 0,Y 587.792,Z 933.38,A -85,B 0,C 180,E1 1358.911,E2 1358.911} C_VEL
LIN {X 0,Y 587.682,Z 905.641,A -85,B 0,C 180,E1 1365.731,E2 1365.731} C_VEL
LIN {X 0,Y 588.265,Z 865.175,A -85,B 0,C 180,E1 1371.763,E2 1371.763} C_VEL
LIN {X 0,Y 589.259,Z 813.714,A -85,B 0,C 180,E1 1376.902,E2 1376.902} C_VEL
LIN {X 0,Y 590.427,Z 753.182,A -85,B 0,C 180,E1 1380.911,E2 1380.911} C_VEL
LIN {X 0,Y 591.308,Z 686.732,A -85,B 0,C 180,E1 1383.488,E2 1383.488} C_VEL
LIN {X 0,Y 589.322,Z 592.075,A -85,B 0,C 180,E1 1385.216,E2 1385.216} C_VEL
LIN {X 0,Y 587.355,Z 586.94,A -85,B 0,C 180,E1 1385.607,E2 1385.607} C_VEL
LIN {X 0,Y 586.286,Z 586.94,A -85,B 0,C 180,E1 1393.307,E2 1393.307} C_VEL
LIN {X 0,Y 586.522,Z 586.94,A -85,B 0,C 180,E1 1399.751,E2 1399.751} C_VEL
LIN {X 0,Y 586.733,Z 586.94,A -85,B 0,C 180,E1 1408.028,E2 1408.028} C_VEL
LIN {X 0,Y 586.445,Z 586.94,A -85,B 0,C 180,E1 1416.723,E2 1416.723} C_VEL
LIN {X 0,Y 587.185,Z 586.94,A -85,B 0,C 180,E1 1424.29,E2 1424.29} C_VEL
LIN {X 0,Y 587,Z 586.94,A -85,B 0,C 180,E1 1433.351,E2 1433.351} C_VEL
LIN {X 0,Y 586.926,Z 586.94,A -85,B 0,C 180,E1 1440.769,E2 1440.769} C_VEL
LIN {X 0,Y 586.79,Z 586.94,A -85,B 0,C 180,E1 1448.203,E2 1448.203} C_VEL
LIN {X 0,Y 586.66,Z 586.94,A -85,B 0,C 180,E1 1455.783,E2 1455.783} C_VEL
LIN {X 0,Y 586.498,Z 586.94,A -85,B 0,C 180,E1 1463.289,E2 1463.289} C_VEL
LIN {X 0,Y 586.523,Z 586.94,A -85,B 0,C 180,E1 1470.319,E2 1470.319} C_VEL
LIN {X 0,Y 587.073,Z 586.94,A -85,B 0,C 180,E1 1477.966,E2 1477.966} C_VEL
LIN {X 0,Y 587.724,Z 588.825,A -85,B 0,C 180,E1 1482.485,E2 1482.485} C_VEL
LIN {X 0,Y 589.13,Z 658.721,A -85,B 0,C 180,E1 1483.843,E2 1483.843} C_VEL
LIN {X 0,Y 588.449,Z 708.916,A -85,B 0,C 180,E1 1486.277,E2 1486.277} C_VEL
LIN {X 0,Y 587.788,Z 752.025,A -85,B 0,C 180,E1 1490.006,E2 1490.006} C_VEL
LIN {X 0,Y 587.325,Z 782.819,A -85,B 0,C 180,E1 1494.494,E2 1494.494} C_VEL
LIN {X 0,Y 587.397,Z 799.757,A -85,B 0,C 180,E1 1498.973,E2 1498.973} C_VEL
LIN {X 0,Y 587.455,Z 805.818,A -85,B 0,C 180,E1 1503.125,E2 1503.125} C_VEL
LIN {X 0,Y 587.563,Z 801.87,A -85,B 0,C 180,E1 1508.008,E2 1508.008} C_VEL
LIN {X 0,Y 587.836,Z 783.324,A -85,B 0,C 180,E1 1513.311,E2 1513.311} C_VEL
LIN {X 0,Y 588.134,Z 751.995,A -85,B 0,C 180,E1 1517.899,E2 1517.899} C_VEL
LIN {X 0,Y 588.58,Z 709.821,A -85,B 0,C 180,E1 1521.568,E2 1521.568} C_VEL
LIN {X 0,Y 589.023,Z 658.298,A -85,B 0,C 180,E1 1524.086,E2 1524.086} C_VEL
LIN {X 0,Y 587.795,Z 589.018,A -85,B 0,C 180,E1 1525.419,E2 1525.419} C_VEL
LIN {X 0,Y 587.182,Z 586.94,A -85,B 0,C 180,E1 1526.296,E2 1526.296} C_VEL
LIN {X 0,Y 586.799,Z 586.94,A -85,B 0,C 180,E1 1533.708,E2 1533.708} C_VEL
LIN {X 0,Y 587.095,Z 586.94,A -85,B 0,C 180,E1 1539.673,E2 1539.673} C_VEL
LIN {X 0,Y 586.862,Z 586.94,A -85,B 0,C 180,E1 1547.3,E2 1547.3} C_VEL
LIN {X 0,Y 586.606,Z 586.94,A -85,B 0,C 180,E1 1555.268,E2 1555.268} C_VEL
LIN {X 0,Y 586.558,Z 586.94,A -85,B 0,C 180,E1 1562.756,E2 1562.756} C_VEL
LIN {X 0,Y 586.65,Z 586.94,A -85,B 0,C 180,E1 1571.272,E2 1571.272} C_VEL
LIN {X 0,Y 587.045,Z 586.94,A -85,B 0,C 180,E1 1578.745,E2 1578.745} C_VEL
LIN {X 0,Y 586.845,Z 586.94,A -85,B 0,C 180,E1 1587.968,E2 1587.968} C_VEL
LIN {X 0,Y 586.499,Z 586.94,A -85,B 0,C 180,E1 1596.714,E2 1596.714} C_VEL
LIN {X 0,Y 587.651,Z 586.94,A -85,B 0,C 180,E1 1605.776,E2 1605.776} C_VEL
LIN {X 0,Y 587.405,Z 586.94,A -85,B 0,C 180,E1 1614.786,E2 1614.786} C_VEL
LIN {X 0,Y 587.279,Z 586.94,A -85,B 0,C 180,E1 1622.192,E2 1622.192} C_VEL
LIN {X 0,Y 587.421,Z 586.94,A -85,B 0,C 180,E1 1628.543,E2 1628.543} C_VEL
LIN {X 0,Y 578.686,Z 586.94,A -85,B 0,C 180,E1 1631.928,E2 1631.928} C_VEL
LIN {X 0,Y 578.551,Z 586.94,A -85,B 0,C 180,E1 1639.101,E2 1639.101} C_VEL
LIN {X 0,Y 578.508,Z 586.94,A -85,B 0,C 180,E1 1645.604,E2 1645.604} C_VEL
LIN {X 0,Y 578.609,Z 586.94,A -85,B 0,C 180,E1 1652.476,E2 1652.476} C_VEL
LIN {X 0,Y 578.523,Z 586.94,A -85,B 0,C 180,E1 1661.618,E2 1661.618} C_VEL
LIN {X 0,Y 578.541,Z 586.94,A -85,B 0,C 180,E1 1670.01,E2 1670.01} C_VEL
LIN {X 0,Y 578.833,Z 588.054,A -85,B 0,C 180,E1 1673.987,E2 1673.987} C_VEL
LIN {X 0,Y 584.334,Z 601.727,A -85,B 0,C 180,E1 1674.581,E2 1674.581} C_VEL
LIN {X 0,Y 584.393,Z 697.179,A -85,B 0,C 180,E1 1676.362,E2 1676.362} C_VEL
LIN {X 0,Y 583.061,Z 763.013,A -85,B 0,C 180,E1 1679.212,E2 1679.212} C_VEL
LIN {X 0,Y 581.592,Z 822.587,A -85,B 0,C 180,E1 1683.485,E2 1683.485} C_VEL
LIN {X 0,Y 580.349,Z 872.146,A -85,B 0,C 180,E1 1688.809,E2 1688.809} C_VEL
LIN {X 0,Y 579.605,Z 910.676,A -85,B 0,C 180,E1 1695.036,E2 1695.036} C_VEL
LIN {X 0,Y 579.38,Z 933.376,A -85,B 0,C 180,E1 1700.958,E2 1700.958} C_VEL
LIN {X 0,Y 579.638,Z 943.766,A -85,B 0,C 180,E1 1706.247,E2 1706.247} C_VEL
LIN {X 0,Y 579.566,Z 945.149,A -85,B 0,C 180,E1 1712.25,E2 1712.25} C_VEL
LIN {X 0,Y 579.749,Z 933.38,A -85,B 0,C 180,E1 1719.035,E2 1719.035} C_VEL
LIN {X 0,Y 579.715,Z 905.643,A -85,B 0,C 180,E1 1725.953,E2 1725.953} C_VEL
LIN {X 0,Y 580.524,Z 864.619,A -85,B 0,C 180,E1 1732.139,E2 1732.139} C_VEL
LIN {X 0,Y 581.883,Z 812.313,A -85,B 0,C 180,E1 1737.388,E2 1737.388} C_VEL
LIN {X 0,Y 583.445,Z 751.735,A -85,B 0,C 180,E1 1741.397,E2 1741.397} C_VEL
LIN {X 0,Y 584.614,Z 686.731,A -85,B 0,C 180,E1 1743.923,E2 1743.923} C_VEL
LIN {X 0,Y 582.843,Z 595.515,A -85,B 0,C 180,E1 1745.616,E2 1745.616} C_VEL
LIN {X 0,Y 579.283,Z 586.94,A -85,B 0,C 180,E1 1746.115,E2 1746.115} C_VEL
LIN {X 0,Y 578.322,Z 586.94,A -85,B 0,C 180,E1 1754.055,E2 1754.055} C_VEL
LIN {X 0,Y 578.196,Z 586.94,A -85,B 0,C 180,E1 1760.736,E2 1760.736} C_VEL
LIN {X 0,Y 578.577,Z 586.94,A -85,B 0,C 180,E1 1768.475,E2 1768.475} C_VEL
LIN {X 0,Y 578.621,Z 586.94,A -85,B 0,C 180,E1 1776.056,E2 1776.056} C_VEL
LIN {X 0,Y 579.147,Z 586.94,A -85,B 0,C 180,E1 1784.067,E2 1784.067} C_VEL
LIN {X 0,Y 579.02,Z 586.94,A -85,B 0,C 180,E1 1793.258,E2 1793.258} C_VEL
LIN {X 0,Y 578.947,Z 586.94,A -85,B 0,C 180,E1 1800.779,E2 1800.779} C_VEL
LIN {X 0,Y 578.766,Z 586.94,A -85,B 0,C 180,E1 1808.317,E2 1808.317} C_VEL
LIN {X 0,Y 578.63,Z 586.94,A -85,B 0,C 180,E1 1816.008,E2 1816.008} C_VEL
LIN {X 0,Y 578.725,Z 586.94,A -85,B 0,C 180,E1 1822.369,E2 1822.369} C_VEL
LIN {X 0,Y 578.389,Z 586.94,A -85,B 0,C 180,E1 1830.792,E2 1830.792} C_VEL
LIN {X 0,Y 578.858,Z 586.94,A -85,B 0,C 180,E1 1839.344,E2 1839.344} C_VEL
LIN {X 0,Y 579.535,Z 588.583,A -85,B 0,C 180,E1 1842.163,E2 1842.163} C_VEL
LIN {X 0,Y 581.605,Z 657.795,A -85,B 0,C 180,E1 1843.539,E2 1843.539} C_VEL
LIN {X 0,Y 580.773,Z 708.987,A -85,B 0,C 180,E1 1846.04,E2 1846.04} C_VEL
LIN {X 0,Y 579.943,Z 752.329,A -85,B 0,C 180,E1 1849.847,E2 1849.847} C_VEL
LIN {X 0,Y 579.32,Z 784.01,A -85,B 0,C 180,E1 1854.594,E2 1854.594} C_VEL
LIN {X 0,Y 579.106,Z 801.445,A -85,B 0,C 180,E1 1859.637,E2 1859.637} C_VEL
LIN {X 0,Y 579.165,Z 805.838,A -85,B 0,C 180,E1 1864.703,E2 1864.703} C_VEL
LIN {X 0,Y 579.304,Z 797.504,A -85,B 0,C 180,E1 1869.843,E2 1869.843} C_VEL
LIN {X 0,Y 579.53,Z 774.672,A -85,B 0,C 180,E1 1875.015,E2 1875.015} C_VEL
LIN {X 0,Y 580.143,Z 738.605,A -85,B 0,C 180,E1 1879.497,E2 1879.497} C_VEL
LIN {X 0,Y 581.098,Z 692.422,A -85,B 0,C 180,E1 1882.87,E2 1882.87} C_VEL
LIN {X 0,Y 581.847,Z 639.753,A -85,B 0,C 180,E1 1884.877,E2 1884.877} C_VEL
LIN {X 0,Y 579.67,Z 588.98,A -85,B 0,C 180,E1 1885.736,E2 1885.736} C_VEL
LIN {X 0,Y 578.946,Z 586.94,A -85,B 0,C 180,E1 1887.747,E2 1887.747} C_VEL
LIN {X 0,Y 578.809,Z 586.94,A -85,B 0,C 180,E1 1895.266,E2 1895.266} C_VEL
LIN {X 0,Y 578.794,Z 586.94,A -85,B 0,C 180,E1 1902.878,E2 1902.878} C_VEL
LIN {X 0,Y 578.792,Z 586.94,A -85,B 0,C 180,E1 1910.73,E2 1910.73} C_VEL
LIN {X 0,Y 578.882,Z 586.94,A -85,B 0,C 180,E1 1919.011,E2 1919.011} C_VEL
LIN {X 0,Y 579.033,Z 586.94,A -85,B 0,C 180,E1 1929.347,E2 1929.347} C_VEL
LIN {X 0,Y 579.151,Z 586.94,A -85,B 0,C 180,E1 1938.312,E2 1938.312} C_VEL
LIN {X 0,Y 578.668,Z 586.94,A -85,B 0,C 180,E1 1948.463,E2 1948.463} C_VEL
LIN {X 0,Y 578.727,Z 586.94,A -85,B 0,C 180,E1 1955.998,E2 1955.998} C_VEL
LIN {X 0,Y 579.651,Z 586.94,A -85,B 0,C 180,E1 1965.575,E2 1965.575} C_VEL
LIN {X 0,Y 579.403,Z 586.94,A -85,B 0,C 180,E1 1974.714,E2 1974.714} C_VEL
LIN {X 0,Y 579.287,Z 586.94,A -85,B 0,C 180,E1 1982.222,E2 1982.222} C_VEL
LIN {X 0,Y 578.817,Z 586.94,A -85,B 0,C 180,E1 1990.526,E2 1990.526} C_VEL
LIN {X 0,Y 578.686,Z 586.94,A -85,B 0,C 180,E1 1991.928,E2 1991.928} C_VEL
LIN {X 0,Y 571.168,Z 586.94,A -85,B 0,C 180,E1 1995.402,E2 1995.402} C_VEL
LIN {X 0,Y 570.918,Z 586.94,A -85,B 0,C 180,E1 2004.288,E2 2004.288} C_VEL
LIN {X 0,Y 570.397,Z 586.94,A -85,B 0,C 180,E1 2013.064,E2 2013.064} C_VEL
LIN {X 0,Y 570.673,Z 586.94,A -85,B 0,C 180,E1 2020.723,E2 2020.723} C_VEL
LIN {X 0,Y 570.701,Z 586.94,A -85,B 0,C 180,E1 2029.347,E2 2029.347} C_VEL
LIN {X 0,Y 570.671,Z 588.384,A -85,B 0,C 180,E1 2033.394,E2 2033.394} C_VEL
LIN {X 0,Y 577.844,Z 605.168,A -85,B 0,C 180,E1 2034.173,E2 2034.173} C_VEL
LIN {X 0,Y 577.642,Z 697.97,A -85,B 0,C 180,E1 2035.942,E2 2035.942} C_VEL
LIN {X 0,Y 575.983,Z 763.881,A -85,B 0,C 180,E1 2038.842,E2 2038.842} C_VEL
LIN {X 0,Y 574.162,Z 822.301,A -85,B 0,C 180,E1 2043.088,E2 2043.088} C_VEL
LIN {X 0,Y 572.662,Z 872.533,A -85,B 0,C 180,E1 2048.564,E2 2048.564} C_VEL
LIN {X 0,Y 571.678,Z 911.549,A -85,B 0,C 180,E1 2055,E2 2055} C_VEL
LIN {X 0,Y 571.067,Z 935.353,A -85,B 0,C 180,E1 2061.595,E2 2061.595} C_VEL
LIN {X 0,Y 570.978,Z 945.148,A -85,B 0,C 180,E1 2067.715,E2 2067.715} C_VEL
LIN {X 0,Y 571.226,Z 943.767,A -85,B 0,C 180,E1 2073.807,E2 2073.807} C_VEL
LIN {X 0,Y 571.207,Z 929.575,A -85,B 0,C 180,E1 2080.443,E2 2080.443} C_VEL
LIN {X 0,Y 571.572,Z 902.534,A -85,B 0,C 180,E1 2086.771,E2 2086.771} C_VEL
LIN {X 0,Y 572.775,Z 862.069,A -85,B 0,C 180,E1 2092.779,E2 2092.779} C_VEL
LIN {X 0,Y 574.642,Z 807.985,A -85,B 0,C 180,E1 2098.13,E2 2098.13} C_VEL
LIN {X 0,Y 576.625,Z 747.237,A -85,B 0,C 180,E1 2102.047,E2 2102.047} C_VEL
LIN {X 0,Y 578.077,Z 683.675,A -85,B 0,C 180,E1 2104.448,E2 2104.448} C_VEL
LIN {X 0,Y 576.222,Z 597.953,A -85,B 0,C 180,E1 2106.052,E2 2106.052} C_VEL
LIN {X 0,Y 571.238,Z 586.94,A -85,B 0,C 180,E1 2106.706,E2 2106.706} C_VEL
LIN {X 0,Y 570.941,Z 586.94,A -85,B 0,C 180,E1 2117.391,E2 2117.391} C_VEL
LIN {X 0,Y 570.792,Z 586.94,A -85,B 0,C 180,E1 2127.024,E2 2127.024} C_VEL
LIN {X 0,Y 570.73,Z 586.94,A -85,B 0,C 180,E1 2135.703,E2 2135.703} C_VEL
LIN {X 0,Y 570.778,Z 586.94,A -85,B 0,C 180,E1 2145.406,E2 2145.406} C_VEL
LIN {X 0,Y 571.035,Z 586.94,A -85,B 0,C 180,E1 2153.164,E2 2153.164} C_VEL
LIN {X 0,Y 570.942,Z 586.94,A -85,B 0,C 180,E1 2160.79,E2 2160.79} C_VEL
LIN {X 0,Y 570.753,Z 586.94,A -85,B 0,C 180,E1 2168.435,E2 2168.435} C_VEL
LIN {X 0,Y 570.613,Z 586.94,A -85,B 0,C 180,E1 2176.239,E2 2176.239} C_VEL
LIN {X 0,Y 570.436,Z 586.94,A -85,B 0,C 180,E1 2184.374,E2 2184.374} C_VEL
LIN {X 0,Y 570.302,Z 586.94,A -85,B 0,C 180,E1 2191.277,E2 2191.277} C_VEL
LIN {X 0,Y 570.94,Z 586.94,A -85,B 0,C 180,E1 2198.673,E2 2198.673} C_VEL
LIN {X 0,Y 571.223,Z 587.253,A -85,B 0,C 180,E1 2201.812,E2 2201.812} C_VEL
LIN {X 0,Y 574.361,Z 615.324,A -85,B 0,C 180,E1 2202.31,E2 2202.31} C_VEL
LIN {X 0,Y 573.913,Z 669.328,A -85,B 0,C 180,E1 2203.687,E2 2203.687} C_VEL
LIN {X 0,Y 572.778,Z 719.216,A -85,B 0,C 180,E1 2206.528,E2 2206.528} C_VEL
LIN {X 0,Y 571.798,Z 759.53,A -85,B 0,C 180,E1 2210.529,E2 2210.529} C_VEL
LIN {X 0,Y 571.191,Z 787.259,A -85,B 0,C 180,E1 2215.167,E2 2215.167} C_VEL
LIN {X 0,Y 571.074,Z 801.788,A -85,B 0,C 180,E1 2219.745,E2 2219.745} C_VEL
LIN {X 0,Y 571.189,Z 805.996,A -85,B 0,C 180,E1 2224.001,E2 2224.001} C_VEL
LIN {X 0,Y 571.448,Z 798.945,A -85,B 0,C 180,E1 2229.399,E2 2229.399} C_VEL
LIN {X 0,Y 571.65,Z 777.896,A -85,B 0,C 180,E1 2234.606,E2 2234.606} C_VEL
LIN {X 0,Y 572.3,Z 743.923,A -85,B 0,C 180,E1 2239.176,E2 2239.176} C_VEL
LIN {X 0,Y 573.392,Z 698.849,A -85,B 0,C 180,E1 2242.757,E2 2242.757} C_VEL
LIN {X 0,Y 574.257,Z 647.077,A -85,B 0,C 180,E1 2244.979,E2 2244.979} C_VEL
LIN {X 0,Y 572.262,Z 590.761,A -85,B 0,C 180,E1 2246.009,E2 2246.009} C_VEL
LIN {X 0,Y 571.224,Z 586.94,A -85,B 0,C 180,E1 2246.193,E2 2246.193} C_VEL
LIN {X 0,Y 570.815,Z 586.94,A -85,B 0,C 180,E1 2253.812,E2 2253.812} C_VEL
LIN {X 0,Y 570.688,Z 586.94,A -85,B 0,C 180,E1 2261.504,E2 2261.504} C_VEL
LIN {X 0,Y 570.617,Z 586.94,A -85,B 0,C 180,E1 2269.417,E2 2269.417} C_VEL
LIN {X 0,Y 570.549,Z 586.94,A -85,B 0,C 180,E1 2277.741,E2 2277.741} C_VEL
LIN {X 0,Y 570.183,Z 586.94,A -85,B 0,C 180,E1 2285.715,E2 2285.715} C_VEL
LIN {X 0,Y 570.302,Z 586.94,A -85,B 0,C 180,E1 2292.949,E2 2292.949} C_VEL
LIN {X 0,Y 570.676,Z 586.94,A -85,B 0,C 180,E1 2299.327,E2 2299.327} C_VEL
LIN {X 0,Y 570.613,Z 586.94,A -85,B 0,C 180,E1 2308.742,E2 2308.742} C_VEL
LIN {X 0,Y 570.462,Z 586.94,A -85,B 0,C 180,E1 2316.602,E2 2316.602} C_VEL
LIN {X 0,Y 571.625,Z 586.94,A -85,B 0,C 180,E1 2325.695,E2 2325.695} C_VEL
LIN {X 0,Y 571.322,Z 586.94,A -85,B 0,C 180,E1 2334.918,E2 2334.918} C_VEL
LIN {X 0,Y 571.267,Z 586.94,A -85,B 0,C 180,E1 2342.254,E2 2342.254} C_VEL
LIN {X 0,Y 571.011,Z 586.94,A -85,B 0,C 180,E1 2349.914,E2 2349.914} C_VEL
LIN {X 0,Y 571.168,Z 586.94,A -85,B 0,C 180,E1 2355.402,E2 2355.402} C_VEL
LIN {X 0,Y 562.561,Z 586.94,A -85,B 0,C 180,E1 2358.886,E2 2358.886} C_VEL
LIN {X 0,Y 562.411,Z 586.94,A -85,B 0,C 180,E1 2366.392,E2 2366.392} C_VEL
LIN {X 0,Y 562.125,Z 586.94,A -85,B 0,C 180,E1 2374.574,E2 2374.574} C_VEL
LIN {X 0,Y 562.36,Z 586.94,A -85,B 0,C 180,E1 2382.09,E2 2382.09} C_VEL
LIN {X 0,Y 562.37,Z 586.94,A -85,B 0,C 180,E1 2390.644,E2 2390.644} C_VEL
LIN {X 0,Y 562.645,Z 588.882,A -85,B 0,C 180,E1 2392.793,E2 2392.793} C_VEL
LIN {X 0,Y 571.401,Z 609.23,A -85,B 0,C 180,E1 2393.768,E2 2393.768} C_VEL
LIN {X 0,Y 570.928,Z 699.065,A -85,B 0,C 180,E1 2395.524,E2 2395.524} C_VEL
LIN {X 0,Y 568.918,Z 765.641,A -85,B 0,C 180,E1 2398.515,E2 2398.515} C_VEL
LIN {X 0,Y 566.67,Z 824.595,A -85,B 0,C 180,E1 2402.918,E2 2402.918} C_VEL
LIN {X 0,Y 564.836,Z 874.169,A -85,B 0,C 180,E1 2408.481,E2 2408.481} C_VEL
LIN {X 0,Y 563.809,Z 911.548,A -85,B 0,C 180,E1 2414.785,E2 2414.785} C_VEL
LIN {X 0,Y 563.117,Z 935.353,A -85,B 0,C 180,E1 2421.476,E2 2421.476} C_VEL
LIN {X 0,Y 562.987,Z 945.149,A -85,B 0,C 180,E1 2427.682,E2 2427.682} C_VEL
LIN {X 0,Y 563.016,Z 943.175,A -85,B 0,C 180,E1 2434.397,E2 2434.397} C_VEL
LIN {X 0,Y 563.168,Z 929.274,A -85,B 0,C 180,E1 2440.696,E2 2440.696} C_VEL
LIN {X 0,Y 563.663,Z 903.463,A -85,B 0,C 180,E1 2446.841,E2 2446.841} C_VEL
LIN {X 0,Y 565.077,Z 862.227,A -85,B 0,C 180,E1 2453.087,E2 2453.087} C_VEL
LIN {X 0,Y 567.299,Z 808.031,A -85,B 0,C 180,E1 2458.524,E2 2458.524} C_VEL
LIN {X 0,Y 569.705,Z 746.573,A -85,B 0,C 180,E1 2462.52,E2 2462.52} C_VEL
LIN {X 0,Y 571.495,Z 682.791,A -85,B 0,C 180,E1 2464.928,E2 2464.928} C_VEL
LIN {X 0,Y 570.035,Z 601.56,A -85,B 0,C 180,E1 2466.451,E2 2466.451} C_VEL
LIN {X 0,Y 563.157,Z 586.94,A -85,B 0,C 180,E1 2467.43,E2 2467.43} C_VEL
LIN {X 0,Y 562.809,Z 586.94,A -85,B 0,C 180,E1 2477.858,E2 2477.858} C_VEL
LIN {X 0,Y 562.527,Z 586.94,A -85,B 0,C 180,E1 2488.31,E2 2488.31} C_VEL
LIN {X 0,Y 562.283,Z 586.94,A -85,B 0,C 180,E1 2497.004,E2 2497.004} C_VEL
LIN {X 0,Y 562.802,Z 586.94,A -85,B 0,C 180,E1 2505.195,E2 2505.195} C_VEL
LIN {X 0,Y 563.046,Z 586.94,A -85,B 0,C 180,E1 2513.066,E2 2513.066} C_VEL
LIN {X 0,Y 562.944,Z 586.94,A -85,B 0,C 180,E1 2520.801,E2 2520.801} C_VEL
LIN {X 0,Y 562.734,Z 586.94,A -85,B 0,C 180,E1 2528.556,E2 2528.556} C_VEL
LIN {X 0,Y 562.624,Z 586.94,A -85,B 0,C 180,E1 2536.764,E2 2536.764} C_VEL
LIN {X 0,Y 562.508,Z 586.94,A -85,B 0,C 180,E1 2545.346,E2 2545.346} C_VEL
LIN {X 0,Y 562.395,Z 586.94,A -85,B 0,C 180,E1 2553.604,E2 2553.604} C_VEL
LIN {X 0,Y 563.257,Z 588.58,A -85,B 0,C 180,E1 2561.5,E2 2561.5} C_VEL
LIN {X 0,Y 566.838,Z 609.556,A -85,B 0,C 180,E1 2561.93,E2 2561.93} C_VEL
LIN {X 0,Y 566.471,Z 666.842,A -85,B 0,C 180,E1 2563.305,E2 2563.305} C_VEL
LIN {X 0,Y 565.102,Z 717.706,A -85,B 0,C 180,E1 2566.164,E2 2566.164} C_VEL
LIN {X 0,Y 563.926,Z 758.95,A -85,B 0,C 180,E1 2570.26,E2 2570.26} C_VEL
LIN {X 0,Y 563.24,Z 786.966,A -85,B 0,C 180,E1 2574.976,E2 2574.976} C_VEL
LIN {X 0,Y 563.019,Z 802.593,A -85,B 0,C 180,E1 2580.091,E2 2580.091} C_VEL
LIN {X 0,Y 563.038,Z 805.541,A -85,B 0,C 180,E1 2585.307,E2 2585.307} C_VEL
LIN {X 0,Y 563.194,Z 796.602,A -85,B 0,C 180,E1 2590.318,E2 2590.318} C_VEL
LIN {X 0,Y 563.646,Z 774.484,A -85,B 0,C 180,E1 2595.361,E2 2595.361} C_VEL
LIN {X 0,Y 564.493,Z 738.626,A -85,B 0,C 180,E1 2599.937,E2 2599.937} C_VEL
LIN {X 0,Y 565.834,Z 692.513,A -85,B 0,C 180,E1 2603.395,E2 2603.395} C_VEL
LIN {X 0,Y 566.881,Z 640.302,A -85,B 0,C 180,E1 2605.442,E2 2605.442} C_VEL
LIN {X 0,Y 564.791,Z 592.67,A -85,B 0,C 180,E1 2606.291,E2 2606.291} C_VEL
LIN {X 0,Y 563.147,Z 586.94,A -85,B 0,C 180,E1 2606.525,E2 2606.525} C_VEL
LIN {X 0,Y 562.825,Z 586.94,A -85,B 0,C 180,E1 2613.866,E2 2613.866} C_VEL
LIN {X 0,Y 562.684,Z 586.94,A -85,B 0,C 180,E1 2621.67,E2 2621.67} C_VEL
LIN {X 0,Y 562.628,Z 586.94,A -85,B 0,C 180,E1 2629.704,E2 2629.704} C_VEL
LIN {X 0,Y 562.586,Z 586.94,A -85,B 0,C 180,E1 2638.168,E2 2638.168} C_VEL
LIN {X 0,Y 562.516,Z 586.94,A -85,B 0,C 180,E1 2647.373,E2 2647.373} C_VEL
LIN {X 0,Y 562.782,Z 586.94,A -85,B 0,C 180,E1 2656.541,E2 2656.541} C_VEL
LIN {X 0,Y 562.809,Z 586.94,A -85,B 0,C 180,E1 2666.424,E2 2666.424} C_VEL
LIN {X 0,Y 562.828,Z 586.94,A -85,B 0,C 180,E1 2675.275,E2 2675.275} C_VEL
LIN {X 0,Y 563.556,Z 586.94,A -85,B 0,C 180,E1 2685.154,E2 2685.154} C_VEL
LIN {X 0,Y 563.395,Z 586.94,A -85,B 0,C 180,E1 2694.563,E2 2694.563} C_VEL
LIN {X 0,Y 563.258,Z 586.94,A -85,B 0,C 180,E1 2702.286,E2 2702.286} C_VEL
LIN {X 0,Y 562.903,Z 586.94,A -85,B 0,C 180,E1 2710.261,E2 2710.261} C_VEL
LIN {X 0,Y 562.648,Z 586.94,A -85,B 0,C 180,E1 2718.031,E2 2718.031} C_VEL
LIN {X 0,Y 562.561,Z 586.94,A -85,B 0,C 180,E1 2718.886,E2 2718.886} C_VEL
LIN {X 0,Y 554.907,Z 586.94,A -85,B 0,C 180,E1 2722.434,E2 2722.434} C_VEL
LIN {X 0,Y 554.574,Z 586.94,A -85,B 0,C 180,E1 2732.199,E2 2732.199} C_VEL
LIN {X 0,Y 554.495,Z 586.94,A -85,B 0,C 180,E1 2741.182,E2 2741.182} C_VEL
LIN {X 0,Y 554.474,Z 586.94,A -85,B 0,C 180,E1 2749.971,E2 2749.971} C_VEL
LIN {X 0,Y 554.584,Z 588.993,A -85,B 0,C 180,E1 2752.16,E2 2752.16} C_VEL
LIN {X 0,Y 564.959,Z 611.441,A -85,B 0,C 180,E1 2753.322,E2 2753.322} C_VEL
LIN {X 0,Y 564.269,Z 699.311,A -85,B 0,C 180,E1 2755.068,E2 2755.068} C_VEL
LIN {X 0,Y 561.891,Z 766.355,A -85,B 0,C 180,E1 2758.118,E2 2758.118} C_VEL
LIN {X 0,Y 559.212,Z 825.742,A -85,B 0,C 180,E1 2762.636,E2 2762.636} C_VEL
LIN {X 0,Y 557.134,Z 874.427,A -85,B 0,C 180,E1 2768.205,E2 2768.205} C_VEL
LIN {X 0,Y 555.968,Z 911.547,A -85,B 0,C 180,E1 2774.565,E2 2774.565} C_VEL
LIN {X 0,Y 555.177,Z 935.354,A -85,B 0,C 180,E1 2781.353,E2 2781.353} C_VEL
LIN {X 0,Y 554.993,Z 945.149,A -85,B 0,C 180,E1 2787.649,E2 2787.649} C_VEL
LIN {X 0,Y 555.035,Z 943.219,A -85,B 0,C 180,E1 2794.421,E2 2794.421} C_VEL
LIN {X 0,Y 555.138,Z 929.274,A -85,B 0,C 180,E1 2800.853,E2 2800.853} C_VEL
LIN {X 0,Y 555.725,Z 902.323,A -85,B 0,C 180,E1 2807.303,E2 2807.303} C_VEL
LIN {X 0,Y 557.406,Z 861.361,A -85,B 0,C 180,E1 2813.536,E2 2813.536} C_VEL
LIN {X 0,Y 560.067,Z 806.286,A -85,B 0,C 180,E1 2819.078,E2 2819.078} C_VEL
LIN {X 0,Y 562.892,Z 745.013,A -85,B 0,C 180,E1 2823.047,E2 2823.047} C_VEL
LIN {X 0,Y 564.927,Z 682.789,A -85,B 0,C 180,E1 2825.394,E2 2825.394} C_VEL
LIN {X 0,Y 563.508,Z 604.523,A -85,B 0,C 180,E1 2826.896,E2 2826.896} C_VEL
LIN {X 0,Y 555.055,Z 586.94,A -85,B 0,C 180,E1 2827.962,E2 2827.962} C_VEL
LIN {X 0,Y 554.64,Z 586.94,A -85,B 0,C 180,E1 2838.799,E2 2838.799} C_VEL
LIN {X 0,Y 554.553,Z 586.94,A -85,B 0,C 180,E1 2847.8,E2 2847.8} C_VEL
LIN {X 0,Y 554.335,Z 586.94,A -85,B 0,C 180,E1 2856.655,E2 2856.655} C_VEL
LIN {X 0,Y 554.811,Z 586.94,A -85,B 0,C 180,E1 2864.976,E2 2864.976} C_VEL
LIN {X 0,Y 555.061,Z 586.94,A -85,B 0,C 180,E1 2872.966,E2 2872.966} C_VEL
LIN {X 0,Y 554.938,Z 586.94,A -85,B 0,C 180,E1 2880.813,E2 2880.813} C_VEL
LIN {X 0,Y 554.75,Z 586.94,A -85,B 0,C 180,E1 2888.68,E2 2888.68} C_VEL
LIN {X 0,Y 554.623,Z 586.94,A -85,B 0,C 180,E1 2896.72,E2 2896.72} C_VEL
LIN {X 0,Y 554.478,Z 586.94,A -85,B 0,C 180,E1 2905.123,E2 2905.123} C_VEL
LIN {X 0,Y 554.364,Z 586.94,A -85,B 0,C 180,E1 2913.395,E2 2913.395} C_VEL
LIN {X 0,Y 555.087,Z 587.933,A -85,B 0,C 180,E1 2921.142,E2 2921.142} C_VEL
LIN {X 0,Y 559.417,Z 609.125,A -85,B 0,C 180,E1 2921.617,E2 2921.617} C_VEL
LIN {X 0,Y 558.979,Z 666.599,A -85,B 0,C 180,E1 2923.005,E2 2923.005} C_VEL
LIN {X 0,Y 557.436,Z 717.113,A -85,B 0,C 180,E1 2925.864,E2 2925.864} C_VEL
LIN {X 0,Y 556.107,Z 757.994,A -85,B 0,C 180,E1 2929.939,E2 2929.939} C_VEL
LIN {X 0,Y 555.332,Z 786.408,A -85,B 0,C 180,E1 2934.72,E2 2934.72} C_VEL
LIN {X 0,Y 555.132,Z 801.786,A -85,B 0,C 180,E1 2939.622,E2 2939.622} C_VEL
LIN {X 0,Y 555.069,Z 805.789,A -85,B 0,C 180,E1 2944.929,E2 2944.929} C_VEL
LIN {X 0,Y 555.276,Z 797.719,A -85,B 0,C 180,E1 2950.026,E2 2950.026} C_VEL
LIN {X 0,Y 555.683,Z 776.25,A -85,B 0,C 180,E1 2955.216,E2 2955.216} C_VEL
LIN {X 0,Y 556.622,Z 742.237,A -85,B 0,C 180,E1 2959.793,E2 2959.793} C_VEL
LIN {X 0,Y 558.142,Z 695.804,A -85,B 0,C 180,E1 2963.476,E2 2963.476} C_VEL
LIN {X 0,Y 559.428,Z 642.925,A -85,B 0,C 180,E1 2965.674,E2 2965.674} C_VEL
LIN {X 0,Y 557.526,Z 594.814,A -85,B 0,C 180,E1 2966.569,E2 2966.569} C_VEL
LIN {X 0,Y 555.083,Z 586.94,A -85,B 0,C 180,E1 2966.81,E2 2966.81} C_VEL
LIN {X 0,Y 554.825,Z 586.94,A -85,B 0,C 180,E1 2973.922,E2 2973.922} C_VEL
LIN {X 0,Y 554.684,Z 586.94,A -85,B 0,C 180,E1 2981.841,E2 2981.841} C_VEL
LIN {X 0,Y 554.664,Z 586.94,A -85,B 0,C 180,E1 2989.999,E2 2989.999} C_VEL
LIN {X 0,Y 554.669,Z 586.94,A -85,B 0,C 180,E1 2998.607,E2 2998.607} C_VEL
LIN {X 0,Y 554.615,Z 586.94,A -85,B 0,C 180,E1 3008.738,E2 3008.738} C_VEL
LIN {X 0,Y 554.679,Z 586.94,A -85,B 0,C 180,E1 3018.796,E2 3018.796} C_VEL
LIN {X 0,Y 554.662,Z 586.94,A -85,B 0,C 180,E1 3027.736,E2 3027.736} C_VEL
LIN {X 0,Y 554.403,Z 586.94,A -85,B 0,C 180,E1 3036.593,E2 3036.593} C_VEL
LIN {X 0,Y 555.511,Z 586.94,A -85,B 0,C 180,E1 3046.548,E2 3046.548} C_VEL
LIN {X 0,Y 554.997,Z 586.94,A -85,B 0,C 180,E1 3056.052,E2 3056.052} C_VEL
LIN {X 0,Y 554.831,Z 586.94,A -85,B 0,C 180,E1 3063.889,E2 3063.889} C_VEL
LIN {X 0,Y 554.7,Z 586.94,A -85,B 0,C 180,E1 3071.805,E2 3071.805} C_VEL
LIN {X 0,Y 554.616,Z 586.94,A -85,B 0,C 180,E1 3079.96,E2 3079.96} C_VEL
LIN {X 0,Y 554.907,Z 586.94,A -85,B 0,C 180,E1 3082.434,E2 3082.434} C_VEL
LIN {X 0,Y 546.478,Z 586.94,A -85,B 0,C 180,E1 3086.017,E2 3086.017} C_VEL
LIN {X 0,Y 546.137,Z 586.94,A -85,B 0,C 180,E1 3094.671,E2 3094.671} C_VEL
LIN {X 0,Y 546.265,Z 586.94,A -85,B 0,C 180,E1 3102.829,E2 3102.829} C_VEL
LIN {X 0,Y 546.311,Z 586.94,A -85,B 0,C 180,E1 3111.396,E2 3111.396} C_VEL
LIN {X 0,Y 558.555,Z 614.164,A -85,B 0,C 180,E1 3112.874,E2 3112.874} C_VEL
LIN {X 0,Y 557.609,Z 700.528,A -85,B 0,C 180,E1 3114.632,E2 3114.632} C_VEL
LIN {X 0,Y 554.914,Z 766.373,A -85,B 0,C 180,E1 3117.67,E2 3117.67} C_VEL
LIN {X 0,Y 551.86,Z 825.589,A -85,B 0,C 180,E1 3122.225,E2 3122.225} C_VEL
LIN {X 0,Y 549.439,Z 874.922,A -85,B 0,C 180,E1 3127.955,E2 3127.955} C_VEL
LIN {X 0,Y 548.091,Z 911.545,A -85,B 0,C 180,E1 3134.338,E2 3134.338} C_VEL
LIN {X 0,Y 547.228,Z 935.354,A -85,B 0,C 180,E1 3141.226,E2 3141.226} C_VEL
LIN {X 0,Y 547.011,Z 945.149,A -85,B 0,C 180,E1 3147.614,E2 3147.614} C_VEL
LIN {X 0,Y 547.011,Z 943.219,A -85,B 0,C 180,E1 3154.486,E2 3154.486} C_VEL
LIN {X 0,Y 547.129,Z 928.96,A -85,B 0,C 180,E1 3161.113,E2 3161.113} C_VEL
LIN {X 0,Y 547.806,Z 902.713,A -85,B 0,C 180,E1 3167.486,E2 3167.486} C_VEL
LIN {X 0,Y 549.699,Z 863.547,A -85,B 0,C 180,E1 3173.596,E2 3173.596} C_VEL
LIN {X 0,Y 552.622,Z 810.465,A -85,B 0,C 180,E1 3179.137,E2 3179.137} C_VEL
LIN {X 0,Y 555.837,Z 749.808,A -85,B 0,C 180,E1 3183.258,E2 3183.258} C_VEL
LIN {X 0,Y 558.28,Z 685.611,A -85,B 0,C 180,E1 3185.794,E2 3185.794} C_VEL
LIN {X 0,Y 556.99,Z 607.013,A -85,B 0,C 180,E1 3187.362,E2 3187.362} C_VEL
LIN {X 0,Y 546.988,Z 586.94,A -85,B 0,C 180,E1 3188.624,E2 3188.624} C_VEL
LIN {X 0,Y 546.74,Z 586.94,A -85,B 0,C 180,E1 3197.351,E2 3197.351} C_VEL
LIN {X 0,Y 546.541,Z 586.94,A -85,B 0,C 180,E1 3207.87,E2 3207.87} C_VEL
LIN {X 0,Y 546.42,Z 586.94,A -85,B 0,C 180,E1 3216.296,E2 3216.296} C_VEL
LIN {X 0,Y 546.814,Z 586.94,A -85,B 0,C 180,E1 3224.751,E2 3224.751} C_VEL
LIN {X 0,Y 547.063,Z 586.94,A -85,B 0,C 180,E1 3232.863,E2 3232.863} C_VEL
LIN {X 0,Y 546.949,Z 586.94,A -85,B 0,C 180,E1 3240.825,E2 3240.825} C_VEL
LIN {X 0,Y 546.735,Z 586.94,A -85,B 0,C 180,E1 3248.808,E2 3248.808} C_VEL
LIN {X 0,Y 546.626,Z 586.94,A -85,B 0,C 180,E1 3256.972,E2 3256.972} C_VEL
LIN {X 0,Y 546.508,Z 586.94,A -85,B 0,C 180,E1 3265.52,E2 3265.52} C_VEL
LIN {X 0,Y 546.609,Z 586.94,A -85,B 0,C 180,E1 3275.017,E2 3275.017} C_VEL
LIN {X 0,Y 546.961,Z 587.227,A -85,B 0,C 180,E1 3280.713,E2 3280.713} C_VEL
LIN {X 0,Y 552.034,Z 610,A -85,B 0,C 180,E1 3281.314,E2 3281.314} C_VEL
LIN {X 0,Y 551.467,Z 666.982,A -85,B 0,C 180,E1 3282.722,E2 3282.722} C_VEL
LIN {X 0,Y 549.727,Z 717.66,A -85,B 0,C 180,E1 3285.646,E2 3285.646} C_VEL
LIN {X 0,Y 548.237,Z 758.435,A -85,B 0,C 180,E1 3289.79,E2 3289.79} C_VEL
LIN {X 0,Y 547.39,Z 786.405,A -85,B 0,C 180,E1 3294.584,E2 3294.584} C_VEL
LIN {X 0,Y 547.06,Z 802.701,A -85,B 0,C 180,E1 3300.047,E2 3300.047} C_VEL
LIN {X 0,Y 547.04,Z 805.882,A -85,B 0,C 180,E1 3304.535,E2 3304.535} C_VEL
LIN {X 0,Y 547.374,Z 798.739,A -85,B 0,C 180,E1 3309.725,E2 3309.725} C_VEL
LIN {X 0,Y 547.722,Z 777.334,A -85,B 0,C 180,E1 3315.182,E2 3315.182} C_VEL
LIN {X 0,Y 548.778,Z 743.903,A -85,B 0,C 180,E1 3319.847,E2 3319.847} C_VEL
LIN {X 0,Y 550.463,Z 698.61,A -85,B 0,C 180,E1 3323.587,E2 3323.587} C_VEL
LIN {X 0,Y 551.837,Z 647.594,A -85,B 0,C 180,E1 3325.861,E2 3325.861} C_VEL
LIN {X 0,Y 550.068,Z 596.66,A -85,B 0,C 180,E1 3326.867,E2 3326.867} C_VEL
LIN {X 0,Y 547.002,Z 586.94,A -85,B 0,C 180,E1 3327.359,E2 3327.359} C_VEL
LIN {X 0,Y 546.819,Z 586.94,A -85,B 0,C 180,E1 3333.979,E2 3333.979} C_VEL
LIN {X 0,Y 546.686,Z 586.94,A -85,B 0,C 180,E1 3342.017,E2 3342.017} C_VEL
LIN {X 0,Y 546.679,Z 586.94,A -85,B 0,C 180,E1 3350.304,E2 3350.304} C_VEL
LIN {X 0,Y 546.667,Z 586.94,A -85,B 0,C 180,E1 3359.065,E2 3359.065} C_VEL
LIN {X 0,Y 546.617,Z 586.94,A -85,B 0,C 180,E1 3368.657,E2 3368.657} C_VEL
LIN {X 0,Y 546.794,Z 586.94,A -85,B 0,C 180,E1 3377.347,E2 3377.347} C_VEL
LIN {X 0,Y 546.657,Z 586.94,A -85,B 0,C 180,E1 3387.854,E2 3387.854} C_VEL
LIN {X 0,Y 546.504,Z 586.94,A -85,B 0,C 180,E1 3396.234,E2 3396.234} C_VEL
LIN {X 0,Y 547.524,Z 586.94,A -85,B 0,C 180,E1 3406.348,E2 3406.348} C_VEL
LIN {X 0,Y 547.004,Z 586.94,A -85,B 0,C 180,E1 3415.994,E2 3415.994} C_VEL
LIN {X 0,Y 546.825,Z 586.94,A -85,B 0,C 180,E1 3423.946,E2 3423.946} C_VEL
LIN {X 0,Y 546.697,Z 586.94,A -85,B 0,C 180,E1 3431.98,E2 3431.98} C_VEL
LIN {X 0,Y 546.638,Z 586.94,A -85,B 0,C 180,E1 3440.264,E2 3440.264} C_VEL
LIN {X 0,Y 546.478,Z 586.94,A -85,B 0,C 180,E1 3446.017,E2 3446.017} C_VEL
LIN {X 0,Y 538.594,Z 586.94,A -85,B 0,C 180,E1 3449.666,E2 3449.666} C_VEL
LIN {X 0,Y 538.564,Z 586.94,A -85,B 0,C 180,E1 3459.286,E2 3459.286} C_VEL
LIN {X 0,Y 538.562,Z 586.94,A -85,B 0,C 180,E1 3468.534,E2 3468.534} C_VEL
LIN {X 0,Y 538.551,Z 588.818,A -85,B 0,C 180,E1 3470.819,E2 3470.819} C_VEL
LIN {X 0,Y 552.186,Z 616.27,A -85,B 0,C 180,E1 3472.406,E2 3472.406} C_VEL
LIN {X 0,Y 551.003,Z 700.76,A -85,B 0,C 180,E1 3474.152,E2 3474.152} C_VEL
LIN {X 0,Y 547.953,Z 766.662,A -85,B 0,C 180,E1 3477.226,E2 3477.226} C_VEL
LIN {X 0,Y 544.455,Z 826.373,A -85,B 0,C 180,E1 3481.891,E2 3481.891} C_VEL
LIN {X 0,Y 541.689,Z 875.974,A -85,B 0,C 180,E1 3487.777,E2 3487.777} C_VEL
LIN {X 0,Y 540.063,Z 913.334,A -85,B 0,C 180,E1 3494.517,E2 3494.517} C_VEL
LIN {X 0,Y 539.306,Z 935.354,A -85,B 0,C 180,E1 3501.096,E2 3501.096} C_VEL
LIN {X 0,Y 539.017,Z 945.149,A -85,B 0,C 180,E1 3507.579,E2 3507.579} C_VEL
LIN {X 0,Y 539.179,Z 943.768,A -85,B 0,C 180,E1 3514.034,E2 3514.034} C_VEL
LIN {X 0,Y 539.282,Z 931.073,A -85,B 0,C 180,E1 3520.538,E2 3520.538} C_VEL
LIN {X 0,Y 539.934,Z 905.65,A -85,B 0,C 180,E1 3527.163,E2 3527.163} C_VEL
LIN {X 0,Y 541.949,Z 865.723,A -85,B 0,C 180,E1 3533.659,E2 3533.659} C_VEL
LIN {X 0,Y 545.201,Z 814.122,A -85,B 0,C 180,E1 3539.241,E2 3539.241} C_VEL
LIN {X 0,Y 548.835,Z 754.222,A -85,B 0,C 180,E1 3543.489,E2 3543.489} C_VEL
LIN {X 0,Y 551.548,Z 690.498,A -85,B 0,C 180,E1 3546.149,E2 3546.149} C_VEL
LIN {X 0,Y 550.823,Z 610.494,A -85,B 0,C 180,E1 3547.797,E2 3547.797} C_VEL
LIN {X 0,Y 538.843,Z 586.94,A -85,B 0,C 180,E1 3549.32,E2 3549.32} C_VEL
LIN {X 0,Y 538.509,Z 586.94,A -85,B 0,C 180,E1 3558.591,E2 3558.591} C_VEL
LIN {X 0,Y 538.415,Z 586.94,A -85,B 0,C 180,E1 3568.622,E2 3568.622} C_VEL
LIN {X 0,Y 538.404,Z 586.94,A -85,B 0,C 180,E1 3576.35,E2 3576.35} C_VEL
LIN {X 0,Y 538.809,Z 586.94,A -85,B 0,C 180,E1 3584.519,E2 3584.519} C_VEL
LIN {X 0,Y 539.061,Z 586.94,A -85,B 0,C 180,E1 3592.756,E2 3592.756} C_VEL
LIN {X 0,Y 538.847,Z 586.94,A -85,B 0,C 180,E1 3601.282,E2 3601.282} C_VEL
LIN {X 0,Y 538.743,Z 586.94,A -85,B 0,C 180,E1 3608.94,E2 3608.94} C_VEL
LIN {X 0,Y 538.626,Z 586.94,A -85,B 0,C 180,E1 3617.232,E2 3617.232} C_VEL
LIN {X 0,Y 538.559,Z 586.94,A -85,B 0,C 180,E1 3625.92,E2 3625.92} C_VEL
LIN {X 0,Y 538.645,Z 586.94,A -85,B 0,C 180,E1 3635.3,E2 3635.3} C_VEL
LIN {X 0,Y 538.991,Z 588.296,A -85,B 0,C 180,E1 3640.219,E2 3640.219} C_VEL
LIN {X 0,Y 544.934,Z 610.44,A -85,B 0,C 180,E1 3640.933,E2 3640.933} C_VEL
LIN {X 0,Y 543.979,Z 666.765,A -85,B 0,C 180,E1 3642.399,E2 3642.399} C_VEL
LIN {X 0,Y 542.087,Z 717.155,A -85,B 0,C 180,E1 3645.337,E2 3645.337} C_VEL
LIN {X 0,Y 540.444,Z 758.024,A -85,B 0,C 180,E1 3649.528,E2 3649.528} C_VEL
LIN {X 0,Y 539.515,Z 785.854,A -85,B 0,C 180,E1 3654.317,E2 3654.317} C_VEL
LIN {X 0,Y 539.134,Z 802.39,A -85,B 0,C 180,E1 3659.807,E2 3659.807} C_VEL
LIN {X 0,Y 539.029,Z 805.97,A -85,B 0,C 180,E1 3664.128,E2 3664.128} C_VEL
LIN {X 0,Y 539.301,Z 798.206,A -85,B 0,C 180,E1 3670.032,E2 3670.032} C_VEL
LIN {X 0,Y 539.81,Z 776.473,A -85,B 0,C 180,E1 3675.511,E2 3675.511} C_VEL
LIN {X 0,Y 540.976,Z 741.802,A -85,B 0,C 180,E1 3680.311,E2 3680.311} C_VEL
LIN {X 0,Y 542.967,Z 695.202,A -85,B 0,C 180,E1 3684.082,E2 3684.082} C_VEL
LIN {X 0,Y 544.64,Z 641.572,A -85,B 0,C 180,E1 3686.361,E2 3686.361} C_VEL
LIN {X 0,Y 542.936,Z 598.141,A -85,B 0,C 180,E1 3687.252,E2 3687.252} C_VEL
LIN {X 0,Y 538.994,Z 586.94,A -85,B 0,C 180,E1 3687.781,E2 3687.781} C_VEL
LIN {X 0,Y 538.872,Z 586.94,A -85,B 0,C 180,E1 3695.657,E2 3695.657} C_VEL
LIN {X 0,Y 538.936,Z 586.94,A -85,B 0,C 180,E1 3703.848,E2 3703.848} C_VEL
LIN {X 0,Y 538.845,Z 586.94,A -85,B 0,C 180,E1 3714.102,E2 3714.102} C_VEL
LIN {X 0,Y 538.265,Z 586.94,A -85,B 0,C 180,E1 3723.706,E2 3723.706} C_VEL
LIN {X 0,Y 538.378,Z 586.94,A -85,B 0,C 180,E1 3731.652,E2 3731.652} C_VEL
LIN {X 0,Y 538.228,Z 586.94,A -85,B 0,C 180,E1 3740.838,E2 3740.838} C_VEL
LIN {X 0,Y 538.398,Z 586.94,A -85,B 0,C 180,E1 3749.281,E2 3749.281} C_VEL
LIN {X 0,Y 538.129,Z 586.94,A -85,B 0,C 180,E1 3757.599,E2 3757.599} C_VEL
LIN {X 0,Y 539.495,Z 586.94,A -85,B 0,C 180,E1 3766.141,E2 3766.141} C_VEL
LIN {X 0,Y 539.01,Z 586.94,A -85,B 0,C 180,E1 3775.935,E2 3775.935} C_VEL
LIN {X 0,Y 538.831,Z 586.94,A -85,B 0,C 180,E1 3784.005,E2 3784.005} C_VEL
LIN {X 0,Y 538.699,Z 586.94,A -85,B 0,C 180,E1 3792.161,E2 3792.161} C_VEL
LIN {X 0,Y 538.678,Z 586.94,A -85,B 0,C 180,E1 3800.577,E2 3800.577} C_VEL
LIN {X 0,Y 538.594,Z 586.94,A -85,B 0,C 180,E1 3809.666,E2 3809.666} C_VEL
LIN {X 0,Y 530.228,Z 586.94,A -85,B 0,C 180,E1 3813.381,E2 3813.381} C_VEL
LIN {X 0,Y 530.246,Z 586.94,A -85,B 0,C 180,E1 3822.201,E2 3822.201} C_VEL
LIN {X 0,Y 530.592,Z 588.855,A -85,B 0,C 180,E1 3830.116,E2 3830.116} C_VEL
LIN {X 0,Y 545.872,Z 620.713,A -85,B 0,C 180,E1 3831.967,E2 3831.967} C_VEL
LIN {X 0,Y 544.423,Z 701.971,A -85,B 0,C 180,E1 3833.696,E2 3833.696} C_VEL
LIN {X 0,Y 540.984,Z 768.005,A -85,B 0,C 180,E1 3836.838,E2 3836.838} C_VEL
LIN {X 0,Y 537.089,Z 827.437,A -85,B 0,C 180,E1 3841.578,E2 3841.578} C_VEL
LIN {X 0,Y 534.063,Z 875.974,A -85,B 0,C 180,E1 3847.443,E2 3847.443} C_VEL
LIN {X 0,Y 532.196,Z 913.335,A -85,B 0,C 180,E1 3854.282,E2 3854.282} C_VEL
LIN {X 0,Y 531.356,Z 935.354,A -85,B 0,C 180,E1 3860.962,E2 3860.962} C_VEL
LIN {X 0,Y 531.042,Z 945.149,A -85,B 0,C 180,E1 3867.543,E2 3867.543} C_VEL
LIN {X 0,Y 531.152,Z 943.768,A -85,B 0,C 180,E1 3874.095,E2 3874.095} C_VEL
LIN {X 0,Y 531.264,Z 931.074,A -85,B 0,C 180,E1 3880.699,E2 3880.699} C_VEL
LIN {X 0,Y 532.004,Z 905.651,A -85,B 0,C 180,E1 3887.427,E2 3887.427} C_VEL
LIN {X 0,Y 534.258,Z 866.781,A -85,B 0,C 180,E1 3893.875,E2 3893.875} C_VEL
LIN {X 0,Y 537.863,Z 815.132,A -85,B 0,C 180,E1 3899.586,E2 3899.586} C_VEL
LIN {X 0,Y 541.975,Z 755.013,A -85,B 0,C 180,E1 3903.92,E2 3903.92} C_VEL
LIN {X 0,Y 545.065,Z 690.574,A -85,B 0,C 180,E1 3906.646,E2 3906.646} C_VEL
LIN {X 0,Y 544.347,Z 613.175,A -85,B 0,C 180,E1 3908.283,E2 3908.283} C_VEL
LIN {X 0,Y 530.628,Z 586.94,A -85,B 0,C 180,E1 3910.05,E2 3910.05} C_VEL
LIN {X 0,Y 530.232,Z 586.94,A -85,B 0,C 180,E1 3919.973,E2 3919.973} C_VEL
LIN {X 0,Y 530.382,Z 586.94,A -85,B 0,C 180,E1 3928.092,E2 3928.092} C_VEL
LIN {X 0,Y 530.137,Z 586.94,A -85,B 0,C 180,E1 3937.31,E2 3937.31} C_VEL
LIN {X 0,Y 530.531,Z 586.94,A -85,B 0,C 180,E1 3945.966,E2 3945.966} C_VEL
LIN {X 0,Y 530.836,Z 586.94,A -85,B 0,C 180,E1 3954.291,E2 3954.291} C_VEL
LIN {X 0,Y 530.965,Z 586.94,A -85,B 0,C 180,E1 3960.85,E2 3960.85} C_VEL
LIN {X 0,Y 530.734,Z 586.94,A -85,B 0,C 180,E1 3969.446,E2 3969.446} C_VEL
LIN {X 0,Y 530.637,Z 586.94,A -85,B 0,C 180,E1 3977.5,E2 3977.5} C_VEL
LIN {X 0,Y 530.603,Z 586.94,A -85,B 0,C 180,E1 3986.338,E2 3986.338} C_VEL
LIN {X 0,Y 530.708,Z 586.94,A -85,B 0,C 180,E1 3995.909,E2 3995.909} C_VEL
LIN {X 0,Y 531.065,Z 588.727,A -85,B 0,C 180,E1 3999.709,E2 3999.709} C_VEL
LIN {X 0,Y 538.042,Z 612.156,A -85,B 0,C 180,E1 4000.532,E2 4000.532} C_VEL
LIN {X 0,Y 536.887,Z 668.094,A -85,B 0,C 180,E1 4002.036,E2 4002.036} C_VEL
LIN {X 0,Y 534.49,Z 716.974,A -85,B 0,C 180,E1 4005.029,E2 4005.029} C_VEL
LIN {X 0,Y 532.617,Z 757.901,A -85,B 0,C 180,E1 4009.295,E2 4009.295} C_VEL
LIN {X 0,Y 531.453,Z 787.201,A -85,B 0,C 180,E1 4014.49,E2 4014.49} C_VEL
LIN {X 0,Y 531.125,Z 802.804,A -85,B 0,C 180,E1 4020,E2 4020} C_VEL
LIN {X 0,Y 531.011,Z 805.458,A -85,B 0,C 180,E1 4025.521,E2 4025.521} C_VEL
LIN {X 0,Y 531.243,Z 795.001,A -85,B 0,C 180,E1 4031.256,E2 4031.256} C_VEL
LIN {X 0,Y 532.041,Z 771.297,A -85,B 0,C 180,E1 4036.601,E2 4036.601} C_VEL
LIN {X 0,Y 533.567,Z 734.486,A -85,B 0,C 180,E1 4041.31,E2 4041.31} C_VEL
LIN {X 0,Y 535.979,Z 685.153,A -85,B 0,C 180,E1 4045.026,E2 4045.026} C_VEL
LIN {X 0,Y 537.757,Z 632.904,A -85,B 0,C 180,E1 4046.975,E2 4046.975} C_VEL
LIN {X 0,Y 535.919,Z 600.049,A -85,B 0,C 180,E1 4047.642,E2 4047.642} C_VEL
LIN {X 0,Y 531.008,Z 586.94,A -85,B 0,C 180,E1 4048.361,E2 4048.361} C_VEL
LIN {X 0,Y 531.139,Z 586.94,A -85,B 0,C 180,E1 4057.388,E2 4057.388} C_VEL
LIN {X 0,Y 530.854,Z 586.94,A -85,B 0,C 180,E1 4067.468,E2 4067.468} C_VEL
LIN {X 0,Y 530.522,Z 586.94,A -85,B 0,C 180,E1 4076.32,E2 4076.32} C_VEL
LIN {X 0,Y 530.193,Z 586.94,A -85,B 0,C 180,E1 4085.319,E2 4085.319} C_VEL
LIN {X 0,Y 530.301,Z 586.94,A -85,B 0,C 180,E1 4094.516,E2 4094.516} C_VEL
LIN {X 0,Y 530.296,Z 586.94,A -85,B 0,C 180,E1 4104.059,E2 4104.059} C_VEL
LIN {X 0,Y 530.661,Z 586.94,A -85,B 0,C 180,E1 4113.665,E2 4113.665} C_VEL
LIN {X 0,Y 531.258,Z 586.94,A -85,B 0,C 180,E1 4124.229,E2 4124.229} C_VEL
LIN {X 0,Y 531.337,Z 586.94,A -85,B 0,C 180,E1 4134.234,E2 4134.234} C_VEL
LIN {X 0,Y 531.235,Z 586.94,A -85,B 0,C 180,E1 4142.424,E2 4142.424} C_VEL
LIN {X 0,Y 530.841,Z 586.94,A -85,B 0,C 180,E1 4150.673,E2 4150.673} C_VEL
LIN {X 0,Y 530.569,Z 586.94,A -85,B 0,C 180,E1 4159.162,E2 4159.162} C_VEL
LIN {X 0,Y 530.45,Z 586.94,A -85,B 0,C 180,E1 4168.119,E2 4168.119} C_VEL
LIN {X 0,Y 530.228,Z 586.94,A -85,B 0,C 180,E1 4173.381,E2 4173.381} C_VEL
LIN {X 0,Y 522.212,Z 586.94,A -85,B 0,C 180,E1 4177.125,E2 4177.125} C_VEL
LIN {X 0,Y 522.492,Z 586.94,A -85,B 0,C 180,E1 4186.957,E2 4186.957} C_VEL
LIN {X 0,Y 522.554,Z 588.452,A -85,B 0,C 180,E1 4189.394,E2 4189.394} C_VEL
LIN {X 0,Y 539.582,Z 622.832,A -85,B 0,C 180,E1 4191.478,E2 4191.478} C_VEL
LIN {X 0,Y 537.882,Z 703.58,A -85,B 0,C 180,E1 4193.244,E2 4193.244} C_VEL
LIN {X 0,Y 534.095,Z 768.001,A -85,B 0,C 180,E1 4196.354,E2 4196.354} C_VEL
LIN {X 0,Y 529.869,Z 826.621,A -85,B 0,C 180,E1 4201.071,E2 4201.071} C_VEL
LIN {X 0,Y 526.411,Z 875.972,A -85,B 0,C 180,E1 4207.096,E2 4207.096} C_VEL
LIN {X 0,Y 524.342,Z 913.337,A -85,B 0,C 180,E1 4214.041,E2 4214.041} C_VEL
LIN {X 0,Y 523.421,Z 935.355,A -85,B 0,C 180,E1 4220.824,E2 4220.824} C_VEL
LIN {X 0,Y 523.074,Z 945.149,A -85,B 0,C 180,E1 4227.505,E2 4227.505} C_VEL
LIN {X 0,Y 523.151,Z 943.769,A -85,B 0,C 180,E1 4234.158,E2 4234.158} C_VEL
LIN {X 0,Y 523.24,Z 931.074,A -85,B 0,C 180,E1 4240.865,E2 4240.865} C_VEL
LIN {X 0,Y 524.104,Z 906.716,A -85,B 0,C 180,E1 4247.464,E2 4247.464} C_VEL
LIN {X 0,Y 526.559,Z 868.379,A -85,B 0,C 180,E1 4254.02,E2 4254.02} C_VEL
LIN {X 0,Y 530.574,Z 816.434,A -85,B 0,C 180,E1 4259.911,E2 4259.911} C_VEL
LIN {X 0,Y 535.154,Z 755.568,A -85,B 0,C 180,E1 4264.377,E2 4264.377} C_VEL
LIN {X 0,Y 538.575,Z 691.992,A -85,B 0,C 180,E1 4267.116,E2 4267.116} C_VEL
LIN {X 0,Y 538.012,Z 616.127,A -85,B 0,C 180,E1 4268.768,E2 4268.768} C_VEL
LIN {X 0,Y 522.542,Z 586.94,A -85,B 0,C 180,E1 4270.799,E2 4270.799} C_VEL
LIN {X 0,Y 522.155,Z 586.94,A -85,B 0,C 180,E1 4280.367,E2 4280.367} C_VEL
LIN {X 0,Y 522.259,Z 586.94,A -85,B 0,C 180,E1 4289.487,E2 4289.487} C_VEL
LIN {X 0,Y 521.978,Z 586.94,A -85,B 0,C 180,E1 4298.734,E2 4298.734} C_VEL
LIN {X 0,Y 522.408,Z 586.94,A -85,B 0,C 180,E1 4306.683,E2 4306.683} C_VEL
LIN {X 0,Y 522.853,Z 586.94,A -85,B 0,C 180,E1 4314.204,E2 4314.204} C_VEL
LIN {X 0,Y 522.978,Z 586.94,A -85,B 0,C 180,E1 4320.863,E2 4320.863} C_VEL
LIN {X 0,Y 522.741,Z 586.94,A -85,B 0,C 180,E1 4329.216,E2 4329.216} C_VEL
LIN {X 0,Y 522.639,Z 586.94,A -85,B 0,C 180,E1 4337.777,E2 4337.777} C_VEL
LIN {X 0,Y 522.59,Z 586.94,A -85,B 0,C 180,E1 4347.667,E2 4347.667} C_VEL
LIN {X 0,Y 522.682,Z 586.94,A -85,B 0,C 180,E1 4357.022,E2 4357.022} C_VEL
LIN {X 0,Y 522.889,Z 587.84,A -85,B 0,C 180,E1 4359.145,E2 4359.145} C_VEL
LIN {X 0,Y 531.167,Z 612.278,A -85,B 0,C 180,E1 4360.095,E2 4360.095} C_VEL
LIN {X 0,Y 529.869,Z 668.421,A -85,B 0,C 180,E1 4361.619,E2 4361.619} C_VEL
LIN {X 0,Y 527.308,Z 716.869,A -85,B 0,C 180,E1 4364.602,E2 4364.602} C_VEL
LIN {X 0,Y 524.765,Z 758.452,A -85,B 0,C 180,E1 4369.145,E2 4369.145} C_VEL
LIN {X 0,Y 523.518,Z 787.215,A -85,B 0,C 180,E1 4374.349,E2 4374.349} C_VEL
LIN {X 0,Y 523.232,Z 802.054,A -85,B 0,C 180,E1 4379.5,E2 4379.5} C_VEL
LIN {X 0,Y 523.006,Z 805.719,A -85,B 0,C 180,E1 4385.121,E2 4385.121} C_VEL
LIN {X 0,Y 523.235,Z 796.185,A -85,B 0,C 180,E1 4390.958,E2 4390.958} C_VEL
LIN {X 0,Y 523.992,Z 773.578,A -85,B 0,C 180,E1 4396.396,E2 4396.396} C_VEL
LIN {X 0,Y 525.944,Z 735.072,A -85,B 0,C 180,E1 4401.602,E2 4401.602} C_VEL
LIN {X 0,Y 528.65,Z 688.083,A -85,B 0,C 180,E1 4405.267,E2 4405.267} C_VEL
LIN {X 0,Y 530.685,Z 635.311,A -85,B 0,C 180,E1 4407.337,E2 4407.337} C_VEL
LIN {X 0,Y 528.813,Z 601.799,A -85,B 0,C 180,E1 4408.05,E2 4408.05} C_VEL
LIN {X 0,Y 523.063,Z 586.94,A -85,B 0,C 180,E1 4408.828,E2 4408.828} C_VEL
LIN {X 0,Y 523.134,Z 586.94,A -85,B 0,C 180,E1 4417.501,E2 4417.501} C_VEL
LIN {X 0,Y 522.783,Z 586.94,A -85,B 0,C 180,E1 4427.746,E2 4427.746} C_VEL
LIN {X 0,Y 522.463,Z 586.94,A -85,B 0,C 180,E1 4436.758,E2 4436.758} C_VEL
LIN {X 0,Y 522.204,Z 586.94,A -85,B 0,C 180,E1 4444.519,E2 4444.519} C_VEL
LIN {X 0,Y 522.249,Z 586.94,A -85,B 0,C 180,E1 4453.068,E2 4453.068} C_VEL
LIN {X 0,Y 522.108,Z 586.94,A -85,B 0,C 180,E1 4461.303,E2 4461.303} C_VEL
LIN {X 0,Y 522.325,Z 586.94,A -85,B 0,C 180,E1 4469.417,E2 4469.417} C_VEL
LIN {X 0,Y 522.224,Z 586.94,A -85,B 0,C 180,E1 4476.878,E2 4476.878} C_VEL
LIN {X 0,Y 523.429,Z 586.94,A -85,B 0,C 180,E1 4486.226,E2 4486.226} C_VEL
LIN {X 0,Y 523.039,Z 586.94,A -85,B 0,C 180,E1 4495.81,E2 4495.81} C_VEL
LIN {X 0,Y 522.821,Z 586.94,A -85,B 0,C 180,E1 4504.128,E2 4504.128} C_VEL
LIN {X 0,Y 522.713,Z 586.94,A -85,B 0,C 180,E1 4512.539,E2 4512.539} C_VEL
LIN {X 0,Y 522.701,Z 586.94,A -85,B 0,C 180,E1 4521.236,E2 4521.236} C_VEL
LIN {X 0,Y 522.464,Z 586.94,A -85,B 0,C 180,E1 4531.035,E2 4531.035} C_VEL
LIN {X 0,Y 522.212,Z 586.94,A -85,B 0,C 180,E1 4537.125,E2 4537.125} C_VEL
LIN {X 0,Y 514.295,Z 586.94,A -85,B 0,C 180,E1 4540.963,E2 4540.963} C_VEL
LIN {X 0,Y 514.563,Z 588.101,A -85,B 0,C 180,E1 4548.786,E2 4548.786} C_VEL
LIN {X 0,Y 533.306,Z 626.191,A -85,B 0,C 180,E1 4550.996,E2 4550.996} C_VEL
LIN {X 0,Y 531.389,Z 704.523,A -85,B 0,C 180,E1 4552.756,E2 4552.756} C_VEL
LIN {X 0,Y 527.096,Z 770.216,A -85,B 0,C 180,E1 4556.008,E2 4556.008} C_VEL
LIN {X 0,Y 522.391,Z 829.331,A -85,B 0,C 180,E1 4560.898,E2 4560.898} C_VEL
LIN {X 0,Y 518.509,Z 878.971,A -85,B 0,C 180,E1 4567.194,E2 4567.194} C_VEL
LIN {X 0,Y 516.289,Z 915.098,A -85,B 0,C 180,E1 4574.223,E2 4574.223} C_VEL
LIN {X 0,Y 515.163,Z 937.286,A -85,B 0,C 180,E1 4581.53,E2 4581.53} C_VEL
LIN {X 0,Y 515.079,Z 945.15,A -85,B 0,C 180,E1 4587.466,E2 4587.466} C_VEL
LIN {X 0,Y 515.124,Z 943.769,A -85,B 0,C 180,E1 4594.223,E2 4594.223} C_VEL
LIN {X 0,Y 515.255,Z 931.075,A -85,B 0,C 180,E1 4601.036,E2 4601.036} C_VEL
LIN {X 0,Y 516.177,Z 907.36,A -85,B 0,C 180,E1 4607.598,E2 4607.598} C_VEL
LIN {X 0,Y 518.928,Z 868.377,A -85,B 0,C 180,E1 4614.396,E2 4614.396} C_VEL
LIN {X 0,Y 523.375,Z 816.434,A -85,B 0,C 180,E1 4620.366,E2 4620.366} C_VEL
LIN {X 0,Y 528.404,Z 755.42,A -85,B 0,C 180,E1 4624.888,E2 4624.888} C_VEL
LIN {X 0,Y 532.234,Z 690.918,A -85,B 0,C 180,E1 4627.67,E2 4627.67} C_VEL
LIN {X 0,Y 532.018,Z 619.67,A -85,B 0,C 180,E1 4629.228,E2 4629.228} C_VEL
LIN {X 0,Y 514.468,Z 586.94,A -85,B 0,C 180,E1 4631.296,E2 4631.296} C_VEL
LIN {X 0,Y 514.11,Z 586.94,A -85,B 0,C 180,E1 4640.668,E2 4640.668} C_VEL
LIN {X 0,Y 514.21,Z 586.94,A -85,B 0,C 180,E1 4650.526,E2 4650.526} C_VEL
LIN {X 0,Y 513.976,Z 586.94,A -85,B 0,C 180,E1 4658.439,E2 4658.439} C_VEL
LIN {X 0,Y 514.392,Z 586.94,A -85,B 0,C 180,E1 4667.255,E2 4667.255} C_VEL
LIN {X 0,Y 514.789,Z 586.94,A -85,B 0,C 180,E1 4675.808,E2 4675.808} C_VEL
LIN {X 0,Y 514.983,Z 586.94,A -85,B 0,C 180,E1 4684.255,E2 4684.255} C_VEL
LIN {X 0,Y 514.897,Z 586.94,A -85,B 0,C 180,E1 4694.535,E2 4694.535} C_VEL
LIN {X 0,Y 514.464,Z 586.94,A -85,B 0,C 180,E1 4703.492,E2 4703.492} C_VEL
LIN {X 0,Y 514.29,Z 586.94,A -85,B 0,C 180,E1 4713.108,E2 4713.108} C_VEL
LIN {X 0,Y 515.025,Z 588.857,A -85,B 0,C 180,E1 4718.602,E2 4718.602} C_VEL
LIN {X 0,Y 524.329,Z 614.091,A -85,B 0,C 180,E1 4719.674,E2 4719.674} C_VEL
LIN {X 0,Y 522.774,Z 670.638,A -85,B 0,C 180,E1 4721.278,E2 4721.278} C_VEL
LIN {X 0,Y 519.801,Z 720.191,A -85,B 0,C 180,E1 4724.446,E2 4724.446} C_VEL
LIN {X 0,Y 517.031,Z 760.907,A -85,B 0,C 180,E1 4729.088,E2 4729.088} C_VEL
LIN {X 0,Y 515.384,Z 790.118,A -85,B 0,C 180,E1 4734.96,E2 4734.96} C_VEL
LIN {X 0,Y 515.091,Z 803.523,A -85,B 0,C 180,E1 4740.38,E2 4740.38} C_VEL
LIN {X 0,Y 515.126,Z 804.656,A -85,B 0,C 180,E1 4746.566,E2 4746.566} C_VEL
LIN {X 0,Y 515.612,Z 791.563,A -85,B 0,C 180,E1 4752.545,E2 4752.545} C_VEL
LIN {X 0,Y 517.08,Z 763.62,A -85,B 0,C 180,E1 4758.361,E2 4758.361} C_VEL
LIN {X 0,Y 519.433,Z 725.013,A -85,B 0,C 180,E1 4762.98,E2 4762.98} C_VEL
LIN {X 0,Y 522.154,Z 676.446,A -85,B 0,C 180,E1 4766.304,E2 4766.304} C_VEL
LIN {X 0,Y 524.046,Z 621.448,A -85,B 0,C 180,E1 4768.033,E2 4768.033} C_VEL
LIN {X 0,Y 520.963,Z 602.089,A -85,B 0,C 180,E1 4768.54,E2 4768.54} C_VEL
LIN {X 0,Y 515.15,Z 586.94,A -85,B 0,C 180,E1 4769.368,E2 4769.368} C_VEL
LIN {X 0,Y 515.137,Z 586.94,A -85,B 0,C 180,E1 4779.325,E2 4779.325} C_VEL
LIN {X 0,Y 514.727,Z 586.94,A -85,B 0,C 180,E1 4788.034,E2 4788.034} C_VEL
LIN {X 0,Y 514.467,Z 586.94,A -85,B 0,C 180,E1 4797.208,E2 4797.208} C_VEL
LIN {X 0,Y 514.131,Z 586.94,A -85,B 0,C 180,E1 4805.715,E2 4805.715} C_VEL
LIN {X 0,Y 514.249,Z 586.94,A -85,B 0,C 180,E1 4813.907,E2 4813.907} C_VEL
LIN {X 0,Y 514.113,Z 586.94,A -85,B 0,C 180,E1 4822.741,E2 4822.741} C_VEL
LIN {X 0,Y 514.294,Z 586.94,A -85,B 0,C 180,E1 4830.841,E2 4830.841} C_VEL
LIN {X 0,Y 514.128,Z 586.94,A -85,B 0,C 180,E1 4840.131,E2 4840.131} C_VEL
LIN {X 0,Y 515.234,Z 586.94,A -85,B 0,C 180,E1 4847.21,E2 4847.21} C_VEL
LIN {X 0,Y 515.042,Z 586.94,A -85,B 0,C 180,E1 4855.745,E2 4855.745} C_VEL
LIN {X 0,Y 514.817,Z 586.94,A -85,B 0,C 180,E1 4864.192,E2 4864.192} C_VEL
LIN {X 0,Y 514.732,Z 586.94,A -85,B 0,C 180,E1 4872.736,E2 4872.736} C_VEL
LIN {X 0,Y 514.689,Z 586.94,A -85,B 0,C 180,E1 4881.757,E2 4881.757} C_VEL
LIN {X 0,Y 514.465,Z 586.94,A -85,B 0,C 180,E1 4891.026,E2 4891.026} C_VEL
LIN {X 0,Y 514.295,Z 586.94,A -85,B 0,C 180,E1 4900.963,E2 4900.963} C_VEL
LIN {X 0,Y 506.179,Z 586.94,A -85,B 0,C 180,E1 4904.836,E2 4904.836} C_VEL
LIN {X 0,Y 506.585,Z 588.399,A -85,B 0,C 180,E1 4908.166,E2 4908.166} C_VEL
LIN {X 0,Y 527.091,Z 630.319,A -85,B 0,C 180,E1 4910.518,E2 4910.518} C_VEL
LIN {X 0,Y 524.821,Z 707.489,A -85,B 0,C 180,E1 4912.327,E2 4912.327} C_VEL
LIN {X 0,Y 520.14,Z 772.268,A -85,B 0,C 180,E1 4915.642,E2 4915.642} C_VEL
LIN {X 0,Y 515.077,Z 830.008,A -85,B 0,C 180,E1 4920.518,E2 4920.518} C_VEL
LIN {X 0,Y 510.771,Z 880.056,A -85,B 0,C 180,E1 4927.001,E2 4927.001} C_VEL
LIN {X 0,Y 508.223,Z 916.837,A -85,B 0,C 180,E1 4934.41,E2 4934.41} C_VEL
LIN {X 0,Y 507.215,Z 937.286,A -85,B 0,C 180,E1 4941.396,E2 4941.396} C_VEL
LIN {X 0,Y 507.112,Z 945.15,A -85,B 0,C 180,E1 4947.427,E2 4947.427} C_VEL
LIN {X 0,Y 507.111,Z 943.769,A -85,B 0,C 180,E1 4954.29,E2 4954.29} C_VEL
LIN {X 0,Y 507.241,Z 931.075,A -85,B 0,C 180,E1 4961.212,E2 4961.212} C_VEL
LIN {X 0,Y 508.31,Z 907.359,A -85,B 0,C 180,E1 4967.88,E2 4967.88} C_VEL
LIN {X 0,Y 511.294,Z 868.866,A -85,B 0,C 180,E1 4974.713,E2 4974.713} C_VEL
LIN {X 0,Y 516.204,Z 816.97,A -85,B 0,C 180,E1 4980.781,E2 4980.781} C_VEL
LIN {X 0,Y 521.611,Z 756.56,A -85,B 0,C 180,E1 4985.334,E2 4985.334} C_VEL
LIN {X 0,Y 525.799,Z 692.422,A -85,B 0,C 180,E1 4988.163,E2 4988.163} C_VEL
LIN {X 0,Y 525.633,Z 622.339,A -85,B 0,C 180,E1 4989.752,E2 4989.752} C_VEL
LIN {X 0,Y 506.338,Z 586.94,A -85,B 0,C 180,E1 4991.999,E2 4991.999} C_VEL
LIN {X 0,Y 506.145,Z 586.94,A -85,B 0,C 180,E1 4999.926,E2 4999.926} C_VEL
LIN {X 0,Y 506.253,Z 586.94,A -85,B 0,C 180,E1 5008.681,E2 5008.681} C_VEL
LIN {X 0,Y 505.986,Z 586.94,A -85,B 0,C 180,E1 5018.027,E2 5018.027} C_VEL
LIN {X 0,Y 506.387,Z 586.94,A -85,B 0,C 180,E1 5027.05,E2 5027.05} C_VEL
LIN {X 0,Y 506.791,Z 586.94,A -85,B 0,C 180,E1 5035.741,E2 5035.741} C_VEL
LIN {X 0,Y 506.786,Z 586.94,A -85,B 0,C 180,E1 5042.606,E2 5042.606} C_VEL
LIN {X 0,Y 506.829,Z 586.94,A -85,B 0,C 180,E1 5051.251,E2 5051.251} C_VEL
LIN {X 0,Y 506.734,Z 586.94,A -85,B 0,C 180,E1 5060.171,E2 5060.171} C_VEL
LIN {X 0,Y 506.439,Z 586.94,A -85,B 0,C 180,E1 5069.656,E2 5069.656} C_VEL
LIN {X 0,Y 506.942,Z 588.71,A -85,B 0,C 180,E1 5078.009,E2 5078.009} C_VEL
LIN {X 0,Y 517.522,Z 615.622,A -85,B 0,C 180,E1 5079.236,E2 5079.236} C_VEL
LIN {X 0,Y 515.749,Z 671.735,A -85,B 0,C 180,E1 5080.874,E2 5080.874} C_VEL
LIN {X 0,Y 512.503,Z 721.505,A -85,B 0,C 180,E1 5084.117,E2 5084.117} C_VEL
LIN {X 0,Y 509.475,Z 761.974,A -85,B 0,C 180,E1 5088.801,E2 5088.801} C_VEL
LIN {X 0,Y 507.664,Z 789.48,A -85,B 0,C 180,E1 5094.346,E2 5094.346} C_VEL
LIN {X 0,Y 507.087,Z 803.77,A -85,B 0,C 180,E1 5100.411,E2 5100.411} C_VEL
LIN {X 0,Y 507.045,Z 805.121,A -85,B 0,C 180,E1 5106.17,E2 5106.17} C_VEL
LIN {X 0,Y 507.543,Z 793.78,A -85,B 0,C 180,E1 5112.21,E2 5112.21} C_VEL
LIN {X 0,Y 509.054,Z 768.716,A -85,B 0,C 180,E1 5117.956,E2 5117.956} C_VEL
LIN {X 0,Y 511.608,Z 731.23,A -85,B 0,C 180,E1 5122.808,E2 5122.808} C_VEL
LIN {X 0,Y 514.662,Z 682.792,A -85,B 0,C 180,E1 5126.408,E2 5126.408} C_VEL
LIN {X 0,Y 516.949,Z 629.58,A -85,B 0,C 180,E1 5128.327,E2 5128.327} C_VEL
LIN {X 0,Y 514.905,Z 606.406,A -85,B 0,C 180,E1 5128.865,E2 5128.865} C_VEL
LIN {X 0,Y 507.264,Z 586.94,A -85,B 0,C 180,E1 5129.809,E2 5129.809} C_VEL
LIN {X 0,Y 507.087,Z 586.94,A -85,B 0,C 180,E1 5139.474,E2 5139.474} C_VEL
LIN {X 0,Y 506.598,Z 586.94,A -85,B 0,C 180,E1 5149.304,E2 5149.304} C_VEL
LIN {X 0,Y 506.428,Z 586.94,A -85,B 0,C 180,E1 5157.848,E2 5157.848} C_VEL
LIN {X 0,Y 506.268,Z 586.94,A -85,B 0,C 180,E1 5167.915,E2 5167.915} C_VEL
LIN {X 0,Y 506.37,Z 586.94,A -85,B 0,C 180,E1 5177.577,E2 5177.577} C_VEL
LIN {X 0,Y 506.357,Z 586.94,A -85,B 0,C 180,E1 5188.343,E2 5188.343} C_VEL
LIN {X 0,Y 506.296,Z 586.94,A -85,B 0,C 180,E1 5196.106,E2 5196.106} C_VEL
LIN {X 0,Y 507.246,Z 586.94,A -85,B 0,C 180,E1 5206.485,E2 5206.485} C_VEL
LIN {X 0,Y 507.044,Z 586.94,A -85,B 0,C 180,E1 5215.678,E2 5215.678} C_VEL
LIN {X 0,Y 507.2,Z 586.94,A -85,B 0,C 180,E1 5222.539,E2 5222.539} C_VEL
LIN {X 0,Y 506.76,Z 586.94,A -85,B 0,C 180,E1 5231.186,E2 5231.186} C_VEL
LIN {X 0,Y 506.564,Z 586.94,A -85,B 0,C 180,E1 5240.108,E2 5240.108} C_VEL
LIN {X 0,Y 506.429,Z 586.94,A -85,B 0,C 180,E1 5249.581,E2 5249.581} C_VEL
LIN {X 0,Y 506.286,Z 586.94,A -85,B 0,C 180,E1 5260.152,E2 5260.152} C_VEL
LIN {X 0,Y 506.179,Z 586.94,A -85,B 0,C 180,E1 5264.836,E2 5264.836} C_VEL
LIN {X 0,Y 498.367,Z 586.94,A -85,B 0,C 180,E1 5267.425,E2 5267.425} C_VEL
LIN {X 0,Y 520.918,Z 632.801,A -85,B 0,C 180,E1 5270.002,E2 5270.002} C_VEL
LIN {X 0,Y 518.391,Z 708.874,A -85,B 0,C 180,E1 5271.832,E2 5271.832} C_VEL
LIN {X 0,Y 513.288,Z 773.076,A -85,B 0,C 180,E1 5275.179,E2 5275.179} C_VEL
LIN {X 0,Y 507.722,Z 831.154,A -85,B 0,C 180,E1 5280.182,E2 5280.182} C_VEL
LIN {X 0,Y 503.125,Z 880.59,A -85,B 0,C 180,E1 5286.719,E2 5286.719} C_VEL
LIN {X 0,Y 500.381,Z 916.836,A -85,B 0,C 180,E1 5294.16,E2 5294.16} C_VEL
LIN {X 0,Y 499.254,Z 937.396,A -85,B 0,C 180,E1 5301.31,E2 5301.31} C_VEL
LIN {X 0,Y 499.115,Z 945.149,A -85,B 0,C 180,E1 5307.385,E2 5307.385} C_VEL
LIN {X 0,Y 499.087,Z 943.769,A -85,B 0,C 180,E1 5314.359,E2 5314.359} C_VEL
LIN {X 0,Y 499.258,Z 931.076,A -85,B 0,C 180,E1 5321.394,E2 5321.394} C_VEL
LIN {X 0,Y 500.47,Z 907.096,A -85,B 0,C 180,E1 5328.231,E2 5328.231} C_VEL
LIN {X 0,Y 503.668,Z 869.602,A -85,B 0,C 180,E1 5335.004,E2 5335.004} C_VEL
LIN {X 0,Y 508.988,Z 818.233,A -85,B 0,C 180,E1 5341.139,E2 5341.139} C_VEL
LIN {X 0,Y 514.875,Z 757.61,A -85,B 0,C 180,E1 5345.795,E2 5345.795} C_VEL
LIN {X 0,Y 519.388,Z 694.453,A -85,B 0,C 180,E1 5348.652,E2 5348.652} C_VEL
LIN {X 0,Y 519.387,Z 625.621,A -85,B 0,C 180,E1 5350.239,E2 5350.239} C_VEL
LIN {X 0,Y 498.266,Z 586.94,A -85,B 0,C 180,E1 5352.581,E2 5352.581} C_VEL
LIN {X 0,Y 497.984,Z 586.94,A -85,B 0,C 180,E1 5361.401,E2 5361.401} C_VEL
LIN {X 0,Y 498.218,Z 586.94,A -85,B 0,C 180,E1 5370.235,E2 5370.235} C_VEL
LIN {X 0,Y 498.02,Z 586.94,A -85,B 0,C 180,E1 5379.531,E2 5379.531} C_VEL
LIN {X 0,Y 498.471,Z 586.94,A -85,B 0,C 180,E1 5388.625,E2 5388.625} C_VEL
LIN {X 0,Y 499.133,Z 586.94,A -85,B 0,C 180,E1 5397.42,E2 5397.42} C_VEL
LIN {X 0,Y 498.894,Z 586.94,A -85,B 0,C 180,E1 5407.898,E2 5407.898} C_VEL
LIN {X 0,Y 498.619,Z 586.94,A -85,B 0,C 180,E1 5416.834,E2 5416.834} C_VEL
LIN {X 0,Y 498.443,Z 586.94,A -85,B 0,C 180,E1 5426.223,E2 5426.223} C_VEL
LIN {X 0,Y 498.654,Z 586.94,A -85,B 0,C 180,E1 5437.32,E2 5437.32} C_VEL
LIN {X 0,Y 510.755,Z 617.85,A -85,B 0,C 180,E1 5438.798,E2 5438.798} C_VEL
LIN {X 0,Y 508.734,Z 673.27,A -85,B 0,C 180,E1 5440.48,E2 5440.48} C_VEL
LIN {X 0,Y 505.259,Z 722.536,A -85,B 0,C 180,E1 5443.752,E2 5443.752} C_VEL
LIN {X 0,Y 501.94,Z 763.14,A -85,B 0,C 180,E1 5448.523,E2 5448.523} C_VEL
LIN {X 0,Y 499.873,Z 790.913,A -85,B 0,C 180,E1 5454.227,E2 5454.227} C_VEL
LIN {X 0,Y 499.242,Z 804.634,A -85,B 0,C 180,E1 5460.058,E2 5460.058} C_VEL
LIN {X 0,Y 499.109,Z 806.599,A -85,B 0,C 180,E1 5465.767,E2 5465.767} C_VEL
LIN {X 0,Y 499.588,Z 796.485,A -85,B 0,C 180,E1 5471.829,E2 5471.829} C_VEL
LIN {X 0,Y 501.154,Z 772.381,A -85,B 0,C 180,E1 5477.763,E2 5477.763} C_VEL
LIN {X 0,Y 503.971,Z 734.603,A -85,B 0,C 180,E1 5482.908,E2 5482.908} C_VEL
LIN {X 0,Y 507.316,Z 687.818,A -85,B 0,C 180,E1 5486.571,E2 5486.571} C_VEL
LIN {X 0,Y 509.861,Z 634.715,A -85,B 0,C 180,E1 5488.663,E2 5488.663} C_VEL
LIN {X 0,Y 508.244,Z 609.284,A -85,B 0,C 180,E1 5489.263,E2 5489.263} C_VEL
LIN {X 0,Y 499.441,Z 586.94,A -85,B 0,C 180,E1 5490.459,E2 5490.459} C_VEL
LIN {X 0,Y 499.057,Z 586.94,A -85,B 0,C 180,E1 5499.628,E2 5499.628} C_VEL
LIN {X 0,Y 498.657,Z 586.94,A -85,B 0,C 180,E1 5508.636,E2 5508.636} C_VEL
LIN {X 0,Y 498.41,Z 586.94,A -85,B 0,C 180,E1 5518.161,E2 5518.161} C_VEL
LIN {X 0,Y 498.201,Z 586.94,A -85,B 0,C 180,E1 5528.641,E2 5528.641} C_VEL
LIN {X 0,Y 498.264,Z 586.94,A -85,B 0,C 180,E1 5538.261,E2 5538.261} C_VEL
LIN {X 0,Y 498.289,Z 586.94,A -85,B 0,C 180,E1 5547.77,E2 5547.77} C_VEL
LIN {X 0,Y 498.314,Z 586.94,A -85,B 0,C 180,E1 5555.699,E2 5555.699} C_VEL
LIN {X 0,Y 499.24,Z 586.94,A -85,B 0,C 180,E1 5564.998,E2 5564.998} C_VEL
LIN {X 0,Y 499.044,Z 586.94,A -85,B 0,C 180,E1 5575.609,E2 5575.609} C_VEL
LIN {X 0,Y 499.181,Z 586.94,A -85,B 0,C 180,E1 5582.579,E2 5582.579} C_VEL
LIN {X 0,Y 498.735,Z 586.94,A -85,B 0,C 180,E1 5591.369,E2 5591.369} C_VEL
LIN {X 0,Y 498.549,Z 586.94,A -85,B 0,C 180,E1 5600.446,E2 5600.446} C_VEL
LIN {X 0,Y 498.379,Z 586.94,A -85,B 0,C 180,E1 5610.108,E2 5610.108} C_VEL
LIN {X 0,Y 498.204,Z 586.94,A -85,B 0,C 180,E1 5619.037,E2 5619.037} C_VEL
LIN {X 0,Y 498.367,Z 586.94,A -85,B 0,C 180,E1 5627.425,E2 5627.425} C_VEL
LIN {X 0,Y 503.483,Z 599.578,A -85,B 0,C 180,E1 5628.106,E2 5628.106} C_VEL
LIN {X 0,Y 506.657,Z 619.32,A -85,B 0,C 180,E1 5628.692,E2 5628.692} C_VEL
LIN {X 0,Y 514.31,Z 636.118,A -85,B 0,C 180,E1 5629.556,E2 5629.556} C_VEL
LIN {X 0,Y 512.026,Z 709.482,A -85,B 0,C 180,E1 5631.296,E2 5631.296} C_VEL
LIN {X 0,Y 506.386,Z 774.845,A -85,B 0,C 180,E1 5634.77,E2 5634.77} C_VEL
LIN {X 0,Y 500.369,Z 832.495,A -85,B 0,C 180,E1 5639.859,E2 5639.859} C_VEL
LIN {X 0,Y 495.454,Z 881.075,A -85,B 0,C 180,E1 5646.421,E2 5646.421} C_VEL
LIN {X 0,Y 492.535,Z 916.835,A -85,B 0,C 180,E1 5653.9,E2 5653.9} C_VEL
LIN {X 0,Y 491.267,Z 937.655,A -85,B 0,C 180,E1 5661.308,E2 5661.308} C_VEL
LIN {X 0,Y 491.123,Z 945.149,A -85,B 0,C 180,E1 5667.343,E2 5667.343} C_VEL
LIN {X 0,Y 491.084,Z 943.769,A -85,B 0,C 180,E1 5674.43,E2 5674.43} C_VEL
LIN {X 0,Y 491.272,Z 931.077,A -85,B 0,C 180,E1 5681.582,E2 5681.582} C_VEL
LIN {X 0,Y 492.564,Z 906.954,A -85,B 0,C 180,E1 5688.568,E2 5688.568} C_VEL
LIN {X 0,Y 496.056,Z 870.368,A -85,B 0,C 180,E1 5695.299,E2 5695.299} C_VEL
LIN {X 0,Y 501.847,Z 818.639,A -85,B 0,C 180,E1 5701.589,E2 5701.589} C_VEL
LIN {X 0,Y 508.178,Z 758.672,A -85,B 0,C 180,E1 5706.267,E2 5706.267} C_VEL
LIN {X 0,Y 513.027,Z 695.507,A -85,B 0,C 180,E1 5709.173,E2 5709.173} C_VEL
LIN {X 0,Y 512.555,Z 628.382,A -85,B 0,C 180,E1 5710.674,E2 5710.674} C_VEL
LIN {X 0,Y 490.2,Z 586.94,A -85,B 0,C 180,E1 5713.115,E2 5713.115} C_VEL
LIN {X 0,Y 489.967,Z 586.94,A -85,B 0,C 180,E1 5722.906,E2 5722.906} C_VEL
LIN {X 0,Y 490.271,Z 586.94,A -85,B 0,C 180,E1 5731.901,E2 5731.901} C_VEL
LIN {X 0,Y 490.531,Z 586.94,A -85,B 0,C 180,E1 5742.951,E2 5742.951} C_VEL
LIN {X 0,Y 490.983,Z 586.94,A -85,B 0,C 180,E1 5752.042,E2 5752.042} C_VEL
LIN {X 0,Y 490.987,Z 586.94,A -85,B 0,C 180,E1 5760.919,E2 5760.919} C_VEL
LIN {X 0,Y 490.734,Z 586.94,A -85,B 0,C 180,E1 5769.823,E2 5769.823} C_VEL
LIN {X 0,Y 490.615,Z 586.94,A -85,B 0,C 180,E1 5779.373,E2 5779.373} C_VEL
LIN {X 0,Y 490.442,Z 586.94,A -85,B 0,C 180,E1 5788.685,E2 5788.685} C_VEL
LIN {X 0,Y 490.796,Z 588.723,A -85,B 0,C 180,E1 5796.745,E2 5796.745} C_VEL
LIN {X 0,Y 504.023,Z 619.626,A -85,B 0,C 180,E1 5798.341,E2 5798.341} C_VEL
LIN {X 0,Y 501.751,Z 674.903,A -85,B 0,C 180,E1 5800.08,E2 5800.08} C_VEL
LIN {X 0,Y 497.93,Z 724.469,A -85,B 0,C 180,E1 5803.459,E2 5803.459} C_VEL
LIN {X 0,Y 494.356,Z 764.627,A -85,B 0,C 180,E1 5808.286,E2 5808.286} C_VEL
LIN {X 0,Y 492.12,Z 792.085,A -85,B 0,C 180,E1 5814.027,E2 5814.027} C_VEL
LIN {X 0,Y 491.547,Z 805.057,A -85,B 0,C 180,E1 5819.378,E2 5819.378} C_VEL
LIN {X 0,Y 491.205,Z 807.855,A -85,B 0,C 180,E1 5825.726,E2 5825.726} C_VEL
LIN {X 0,Y 491.784,Z 797.489,A -85,B 0,C 180,E1 5832.028,E2 5832.028} C_VEL
LIN {X 0,Y 493.496,Z 773.423,A -85,B 0,C 180,E1 5838.021,E2 5838.021} C_VEL
LIN {X 0,Y 496.598,Z 735.618,A -85,B 0,C 180,E1 5843.243,E2 5843.243} C_VEL
LIN {X 0,Y 500.307,Z 687.123,A -85,B 0,C 180,E1 5847.067,E2 5847.067} C_VEL
LIN {X 0,Y 503.005,Z 634.224,A -85,B 0,C 180,E1 5849.136,E2 5849.136} C_VEL
LIN {X 0,Y 501.2,Z 611.139,A -85,B 0,C 180,E1 5849.717,E2 5849.717} C_VEL
LIN {X 0,Y 491.559,Z 586.94,A -85,B 0,C 180,E1 5850.885,E2 5850.885} C_VEL
LIN {X 0,Y 490.736,Z 586.94,A -85,B 0,C 180,E1 5861.596,E2 5861.596} C_VEL
LIN {X 0,Y 490.594,Z 586.94,A -85,B 0,C 180,E1 5870.838,E2 5870.838} C_VEL
LIN {X 0,Y 490.33,Z 586.94,A -85,B 0,C 180,E1 5880.709,E2 5880.709} C_VEL
LIN {X 0,Y 490.193,Z 586.94,A -85,B 0,C 180,E1 5890.646,E2 5890.646} C_VEL
LIN {X 0,Y 490.063,Z 586.94,A -85,B 0,C 180,E1 5900.57,E2 5900.57} C_VEL
LIN {X 0,Y 490.23,Z 586.94,A -85,B 0,C 180,E1 5909.26,E2 5909.26} C_VEL
LIN {X 0,Y 490.027,Z 586.94,A -85,B 0,C 180,E1 5919.11,E2 5919.11} C_VEL
LIN {X 0,Y 491.236,Z 586.94,A -85,B 0,C 180,E1 5926.682,E2 5926.682} C_VEL
LIN {X 0,Y 491.043,Z 586.94,A -85,B 0,C 180,E1 5935.537,E2 5935.537} C_VEL
LIN {X 0,Y 491.178,Z 586.94,A -85,B 0,C 180,E1 5942.621,E2 5942.621} C_VEL
LIN {X 0,Y 490.712,Z 586.94,A -85,B 0,C 180,E1 5951.557,E2 5951.557} C_VEL
LIN {X 0,Y 490.552,Z 586.94,A -85,B 0,C 180,E1 5960.795,E2 5960.795} C_VEL
LIN {X 0,Y 490.28,Z 586.94,A -85,B 0,C 180,E1 5970.658,E2 5970.658} C_VEL
LIN {X 0,Y 490.161,Z 586.94,A -85,B 0,C 180,E1 5980.666,E2 5980.666} C_VEL
LIN {X 0,Y 490.324,Z 587.833,A -85,B 0,C 180,E1 5986.802,E2 5986.802} C_VEL
LIN {X 0,Y 506.657,Z 619.32,A -85,B 0,C 180,E1 5988.692,E2 5988.692} C_VEL
LIN {X 0,Y 509.108,Z 636.25,A -85,B 0,C 180,E1 5989.153,E2 5989.153} C_VEL
LIN {X 0,Y 507.677,Z 654.794,A -85,B 0,C 180,E1 5989.367,E2 5989.367} C_VEL
LIN {X 0,Y 504.631,Z 722.863,A -85,B 0,C 180,E1 5991.344,E2 5991.344} C_VEL
LIN {X 0,Y 498.946,Z 782.691,A -85,B 0,C 180,E1 5994.8,E2 5994.8} C_VEL
LIN {X 0,Y 492.221,Z 840.797,A -85,B 0,C 180,E1 6000.316,E2 6000.316} C_VEL
LIN {X 0,Y 486.823,Z 888.378,A -85,B 0,C 180,E1 6007.309,E2 6007.309} C_VEL
LIN {X 0,Y 483.979,Z 921.647,A -85,B 0,C 180,E1 6015.007,E2 6015.007} C_VEL
LIN {X 0,Y 483.064,Z 938.884,A -85,B 0,C 180,E1 6021.872,E2 6021.872} C_VEL
LIN {X 0,Y 483.125,Z 945.149,A -85,B 0,C 180,E1 6027.299,E2 6027.299} C_VEL
LIN {X 0,Y 483.063,Z 943.768,A -85,B 0,C 180,E1 6034.504,E2 6034.504} C_VEL
LIN {X 0,Y 483.293,Z 931.076,A -85,B 0,C 180,E1 6041.776,E2 6041.776} C_VEL
LIN {X 0,Y 484.693,Z 906.746,A -85,B 0,C 180,E1 6048.931,E2 6048.931} C_VEL
LIN {X 0,Y 488.481,Z 870.657,A -85,B 0,C 180,E1 6055.674,E2 6055.674} C_VEL
LIN {X 0,Y 494.788,Z 818.835,A -85,B 0,C 180,E1 6062.07,E2 6062.07} C_VEL
LIN {X 0,Y 501.533,Z 759.304,A -85,B 0,C 180,E1 6066.781,E2 6066.781} C_VEL
LIN {X 0,Y 506.157,Z 696.645,A -85,B 0,C 180,E1 6069.614,E2 6069.614} C_VEL
LIN {X 0,Y 505.988,Z 631.767,A -85,B 0,C 180,E1 6071.097,E2 6071.097} C_VEL
LIN {X 0,Y 482.214,Z 586.94,A -85,B 0,C 180,E1 6073.9,E2 6073.9} C_VEL
LIN {X 0,Y 481.997,Z 586.94,A -85,B 0,C 180,E1 6084.435,E2 6084.435} C_VEL
LIN {X 0,Y 482.21,Z 586.94,A -85,B 0,C 180,E1 6094.908,E2 6094.908} C_VEL
LIN {X 0,Y 482.527,Z 586.94,A -85,B 0,C 180,E1 6104.537,E2 6104.537} C_VEL
LIN {X 0,Y 482.857,Z 586.94,A -85,B 0,C 180,E1 6113.722,E2 6113.722} C_VEL
LIN {X 0,Y 482.981,Z 586.94,A -85,B 0,C 180,E1 6120.934,E2 6120.934} C_VEL
LIN {X 0,Y 482.74,Z 586.94,A -85,B 0,C 180,E1 6129.987,E2 6129.987} C_VEL
LIN {X 0,Y 482.63,Z 586.94,A -85,B 0,C 180,E1 6139.306,E2 6139.306} C_VEL
LIN {X 0,Y 482.333,Z 586.94,A -85,B 0,C 180,E1 6149.214,E2 6149.214} C_VEL
LIN {X 0,Y 482.6,Z 588.219,A -85,B 0,C 180,E1 6156.048,E2 6156.048} C_VEL
LIN {X 0,Y 497.272,Z 622.887,A -85,B 0,C 180,E1 6157.897,E2 6157.897} C_VEL
LIN {X 0,Y 494.756,Z 677.125,A -85,B 0,C 180,E1 6159.696,E2 6159.696} C_VEL
LIN {X 0,Y 490.592,Z 726.543,A -85,B 0,C 180,E1 6163.168,E2 6163.168} C_VEL
LIN {X 0,Y 486.651,Z 767.262,A -85,B 0,C 180,E1 6168.228,E2 6168.228} C_VEL
LIN {X 0,Y 484.203,Z 794.586,A -85,B 0,C 180,E1 6174.232,E2 6174.232} C_VEL
LIN {X 0,Y 483.567,Z 806.831,A -85,B 0,C 180,E1 6179.684,E2 6179.684} C_VEL
LIN {X 0,Y 483.24,Z 809.488,A -85,B 0,C 180,E1 6184.917,E2 6184.917} C_VEL
LIN {X 0,Y 483.794,Z 801.018,A -85,B 0,C 180,E1 6191.246,E2 6191.246} C_VEL
LIN {X 0,Y 485.294,Z 779.273,A -85,B 0,C 180,E1 6197.357,E2 6197.357} C_VEL
LIN {X 0,Y 488.408,Z 744.307,A -85,B 0,C 180,E1 6202.734,E2 6202.734} C_VEL
LIN {X 0,Y 492.553,Z 697.215,A -85,B 0,C 180,E1 6206.91,E2 6206.91} C_VEL
LIN {X 0,Y 495.783,Z 644.111,A -85,B 0,C 180,E1 6209.355,E2 6209.355} C_VEL
LIN {X 0,Y 494.472,Z 613.771,A -85,B 0,C 180,E1 6210.151,E2 6210.151} C_VEL
LIN {X 0,Y 483.35,Z 586.94,A -85,B 0,C 180,E1 6211.575,E2 6211.575} C_VEL
LIN {X 0,Y 482.75,Z 586.94,A -85,B 0,C 180,E1 6221.791,E2 6221.791} C_VEL
LIN {X 0,Y 482.56,Z 586.94,A -85,B 0,C 180,E1 6231.887,E2 6231.887} C_VEL
LIN {X 0,Y 482.293,Z 586.94,A -85,B 0,C 180,E1 6241.277,E2 6241.277} C_VEL
LIN {X 0,Y 482.182,Z 586.94,A -85,B 0,C 180,E1 6250.18,E2 6250.18} C_VEL
LIN {X 0,Y 482.062,Z 586.94,A -85,B 0,C 180,E1 6260.468,E2 6260.468} C_VEL
LIN {X 0,Y 482.224,Z 586.94,A -85,B 0,C 180,E1 6270.779,E2 6270.779} C_VEL
LIN {X 0,Y 482.221,Z 586.94,A -85,B 0,C 180,E1 6280.677,E2 6280.677} C_VEL
LIN {X 0,Y 482.972,Z 586.94,A -85,B 0,C 180,E1 6288.185,E2 6288.185} C_VEL
LIN {X 0,Y 482.821,Z 586.94,A -85,B 0,C 180,E1 6297.264,E2 6297.264} C_VEL
LIN {X 0,Y 482.805,Z 586.94,A -85,B 0,C 180,E1 6304.471,E2 6304.471} C_VEL
LIN {X 0,Y 482.712,Z 586.94,A -85,B 0,C 180,E1 6313.597,E2 6313.597} C_VEL
LIN {X 0,Y 482.565,Z 586.94,A -85,B 0,C 180,E1 6323.1,E2 6323.1} C_VEL
LIN {X 0,Y 482.064,Z 586.94,A -85,B 0,C 180,E1 6333.465,E2 6333.465} C_VEL
LIN {X 0,Y 482.097,Z 586.94,A -85,B 0,C 180,E1 6342.524,E2 6342.524} C_VEL
LIN {X 0,Y 482.486,Z 588.826,A -85,B 0,C 180,E1 6346.125,E2 6346.125} C_VEL
LIN {X 0,Y 507.685,Z 636.886,A -85,B 0,C 180,E1 6349.066,E2 6349.066} C_VEL
LIN {X 0,Y 507.677,Z 654.794,A -85,B 0,C 180,E1 6349.367,E2 6349.367} C_VEL
LIN {X 0,Y 499.714,Z 689.329,A -85,B 0,C 180,E1 6349.641,E2 6349.641} C_VEL
LIN {X 0,Y 495.018,Z 756.611,A -85,B 0,C 180,E1 6352.558,E2 6352.558} C_VEL
LIN {X 0,Y 488.834,Z 810.19,A -85,B 0,C 180,E1 6356.577,E2 6356.577} C_VEL
LIN {X 0,Y 482.11,Z 862.335,A -85,B 0,C 180,E1 6362.653,E2 6362.653} C_VEL
LIN {X 0,Y 477.407,Z 901.836,A -85,B 0,C 180,E1 6369.639,E2 6369.639} C_VEL
LIN {X 0,Y 475.525,Z 928.02,A -85,B 0,C 180,E1 6376.86,E2 6376.86} C_VEL
LIN {X 0,Y 475.123,Z 942.889,A -85,B 0,C 180,E1 6384.501,E2 6384.501} C_VEL
LIN {X 0,Y 475.426,Z 945.15,A -85,B 0,C 180,E1 6392.743,E2 6392.743} C_VEL
LIN {X 0,Y 475.512,Z 935.359,A -85,B 0,C 180,E1 6400.108,E2 6400.108} C_VEL
LIN {X 0,Y 476.606,Z 913.348,A -85,B 0,C 180,E1 6407.606,E2 6407.606} C_VEL
LIN {X 0,Y 480.33,Z 877.043,A -85,B 0,C 180,E1 6415.062,E2 6415.062} C_VEL
LIN {X 0,Y 486.634,Z 828.065,A -85,B 0,C 180,E1 6421.619,E2 6421.619} C_VEL
LIN {X 0,Y 493.611,Z 770.926,A -85,B 0,C 180,E1 6426.563,E2 6426.563} C_VEL
LIN {X 0,Y 498.671,Z 704.72,A -85,B 0,C 180,E1 6429.832,E2 6429.832} C_VEL
LIN {X 0,Y 499.49,Z 635.124,A -85,B 0,C 180,E1 6431.535,E2 6431.535} C_VEL
LIN {X 0,Y 474.164,Z 586.94,A -85,B 0,C 180,E1 6434.577,E2 6434.577} C_VEL
LIN {X 0,Y 473.972,Z 586.94,A -85,B 0,C 180,E1 6444.728,E2 6444.728} C_VEL
LIN {X 0,Y 474.206,Z 586.94,A -85,B 0,C 180,E1 6454.454,E2 6454.454} C_VEL
LIN {X 0,Y 474.505,Z 586.94,A -85,B 0,C 180,E1 6464.269,E2 6464.269} C_VEL
LIN {X 0,Y 474.854,Z 586.94,A -85,B 0,C 180,E1 6473.616,E2 6473.616} C_VEL
LIN {X 0,Y 474.993,Z 586.94,A -85,B 0,C 180,E1 6480.95,E2 6480.95} C_VEL
LIN {X 0,Y 474.729,Z 586.94,A -85,B 0,C 180,E1 6490.157,E2 6490.157} C_VEL
LIN {X 0,Y 474.606,Z 586.94,A -85,B 0,C 180,E1 6499.646,E2 6499.646} C_VEL
LIN {X 0,Y 474.306,Z 586.94,A -85,B 0,C 180,E1 6509.757,E2 6509.757} C_VEL
LIN {X 0,Y 474.444,Z 587.884,A -85,B 0,C 180,E1 6515.328,E2 6515.328} C_VEL
LIN {X 0,Y 490.587,Z 624.208,A -85,B 0,C 180,E1 6517.407,E2 6517.407} C_VEL
LIN {X 0,Y 487.767,Z 679.524,A -85,B 0,C 180,E1 6519.31,E2 6519.31} C_VEL
LIN {X 0,Y 483.24,Z 728.987,A -85,B 0,C 180,E1 6522.903,E2 6522.903} C_VEL
LIN {X 0,Y 479.078,Z 768.87,A -85,B 0,C 180,E1 6527.999,E2 6527.999} C_VEL
LIN {X 0,Y 476.492,Z 795.366,A -85,B 0,C 180,E1 6533.902,E2 6533.902} C_VEL
LIN {X 0,Y 475.547,Z 809.017,A -85,B 0,C 180,E1 6540.356,E2 6540.356} C_VEL
LIN {X 0,Y 475.679,Z 808.98,A -85,B 0,C 180,E1 6547.403,E2 6547.403} C_VEL
LIN {X 0,Y 476.789,Z 794.979,A -85,B 0,C 180,E1 6553.932,E2 6553.932} C_VEL
LIN {X 0,Y 479.198,Z 767.346,A -85,B 0,C 180,E1 6559.97,E2 6559.97} C_VEL
LIN {X 0,Y 482.897,Z 727.845,A -85,B 0,C 180,E1 6564.93,E2 6564.93} C_VEL
LIN {X 0,Y 486.945,Z 679.183,A -85,B 0,C 180,E1 6568.441,E2 6568.441} C_VEL
LIN {X 0,Y 489.687,Z 622.85,A -85,B 0,C 180,E1 6570.333,E2 6570.333} C_VEL
LIN {X 0,Y 475.223,Z 586.94,A -85,B 0,C 180,E1 6572.239,E2 6572.239} C_VEL
LIN {X 0,Y 474.727,Z 586.94,A -85,B 0,C 180,E1 6581.993,E2 6581.993} C_VEL
LIN {X 0,Y 474.556,Z 586.94,A -85,B 0,C 180,E1 6591.577,E2 6591.577} C_VEL
LIN {X 0,Y 474.193,Z 586.94,A -85,B 0,C 180,E1 6601.97,E2 6601.97} C_VEL
LIN {X 0,Y 474.084,Z 586.94,A -85,B 0,C 180,E1 6611.19,E2 6611.19} C_VEL
LIN {X 0,Y 474.026,Z 586.94,A -85,B 0,C 180,E1 6621.345,E2 6621.345} C_VEL
LIN {X 0,Y 474.202,Z 586.94,A -85,B 0,C 180,E1 6631.649,E2 6631.649} C_VEL
LIN {X 0,Y 474.553,Z 586.94,A -85,B 0,C 180,E1 6642.285,E2 6642.285} C_VEL
LIN {X 0,Y 474.781,Z 586.94,A -85,B 0,C 180,E1 6649.844,E2 6649.844} C_VEL
LIN {X 0,Y 475.018,Z 586.94,A -85,B 0,C 180,E1 6659.05,E2 6659.05} C_VEL
LIN {X 0,Y 475.114,Z 586.94,A -85,B 0,C 180,E1 6668.225,E2 6668.225} C_VEL
LIN {X 0,Y 474.641,Z 586.94,A -85,B 0,C 180,E1 6677.638,E2 6677.638} C_VEL
LIN {X 0,Y 474.242,Z 586.94,A -85,B 0,C 180,E1 6687.593,E2 6687.593} C_VEL
LIN {X 0,Y 474.104,Z 586.94,A -85,B 0,C 180,E1 6698.352,E2 6698.352} C_VEL
LIN {X 0,Y 474.414,Z 588.852,A -85,B 0,C 180,E1 6705.384,E2 6705.384} C_VEL
LIN {X 0,Y 501.111,Z 640.79,A -85,B 0,C 180,E1 6708.612,E2 6708.612} C_VEL
LIN {X 0,Y 499.714,Z 689.329,A -85,B 0,C 180,E1 6709.641,E2 6709.641} C_VEL
LIN {X 0,Y 491.588,Z 711.812,A -85,B 0,C 180,E1 6709.882,E2 6709.882} C_VEL
LIN {X 0,Y 485.442,Z 779.732,A -85,B 0,C 180,E1 6713.561,E2 6713.561} C_VEL
LIN {X 0,Y 479.175,Z 831.428,A -85,B 0,C 180,E1 6718.242,E2 6718.242} C_VEL
LIN {X 0,Y 472.736,Z 880.348,A -85,B 0,C 180,E1 6725.082,E2 6725.082} C_VEL
LIN {X 0,Y 468.998,Z 915.984,A -85,B 0,C 180,E1 6732.833,E2 6732.833} C_VEL
LIN {X 0,Y 467.512,Z 937.285,A -85,B 0,C 180,E1 6740.659,E2 6740.659} C_VEL
LIN {X 0,Y 467.134,Z 945.148,A -85,B 0,C 180,E1 6747.206,E2 6747.206} C_VEL
LIN {X 0,Y 467.027,Z 943.768,A -85,B 0,C 180,E1 6754.659,E2 6754.659} C_VEL
LIN {X 0,Y 467.374,Z 931.076,A -85,B 0,C 180,E1 6762.183,E2 6762.183} C_VEL
LIN {X 0,Y 469.011,Z 907.629,A -85,B 0,C 180,E1 6769.368,E2 6769.368} C_VEL
LIN {X 0,Y 473.533,Z 870.836,A -85,B 0,C 180,E1 6776.518,E2 6776.518} C_VEL
LIN {X 0,Y 480.881,Z 818.355,A -85,B 0,C 180,E1 6783.17,E2 6783.17} C_VEL
LIN {X 0,Y 487.255,Z 763.038,A -85,B 0,C 180,E1 6787.508,E2 6787.508} C_VEL
LIN {X 0,Y 492.533,Z 697.115,A -85,B 0,C 180,E1 6790.574,E2 6790.574} C_VEL
LIN {X 0,Y 492.695,Z 637.8,A -85,B 0,C 180,E1 6792.021,E2 6792.021} C_VEL
LIN {X 0,Y 466.142,Z 586.94,A -85,B 0,C 180,E1 6795.388,E2 6795.388} C_VEL
LIN {X 0,Y 466.011,Z 586.94,A -85,B 0,C 180,E1 6806.136,E2 6806.136} C_VEL
LIN {X 0,Y 466.045,Z 586.94,A -85,B 0,C 180,E1 6816.031,E2 6816.031} C_VEL
LIN {X 0,Y 466.406,Z 586.94,A -85,B 0,C 180,E1 6825.918,E2 6825.918} C_VEL
LIN {X 0,Y 466.787,Z 586.94,A -85,B 0,C 180,E1 6835.376,E2 6835.376} C_VEL
LIN {X 0,Y 466.791,Z 586.94,A -85,B 0,C 180,E1 6842.83,E2 6842.83} C_VEL
LIN {X 0,Y 466.826,Z 586.94,A -85,B 0,C 180,E1 6852.23,E2 6852.23} C_VEL
LIN {X 0,Y 466.451,Z 586.94,A -85,B 0,C 180,E1 6862,E2 6862} C_VEL
LIN {X 0,Y 466.144,Z 586.94,A -85,B 0,C 180,E1 6872.518,E2 6872.518} C_VEL
LIN {X 0,Y 466.422,Z 588.499,A -85,B 0,C 180,E1 6874.606,E2 6874.606} C_VEL
LIN {X 0,Y 483.877,Z 627.346,A -85,B 0,C 180,E1 6876.94,E2 6876.94} C_VEL
LIN {X 0,Y 480.804,Z 681.609,A -85,B 0,C 180,E1 6878.899,E2 6878.899} C_VEL
LIN {X 0,Y 475.945,Z 731.077,A -85,B 0,C 180,E1 6882.597,E2 6882.597} C_VEL
LIN {X 0,Y 471.479,Z 770.634,A -85,B 0,C 180,E1 6887.787,E2 6887.787} C_VEL
LIN {X 0,Y 468.703,Z 796.911,A -85,B 0,C 180,E1 6893.807,E2 6893.807} C_VEL
LIN {X 0,Y 467.766,Z 809.678,A -85,B 0,C 180,E1 6899.812,E2 6899.812} C_VEL
LIN {X 0,Y 467.586,Z 811.371,A -85,B 0,C 180,E1 6906.067,E2 6906.067} C_VEL
LIN {X 0,Y 468.487,Z 799.827,A -85,B 0,C 180,E1 6912.901,E2 6912.901} C_VEL
LIN {X 0,Y 470.915,Z 774.46,A -85,B 0,C 180,E1 6919.218,E2 6919.218} C_VEL
LIN {X 0,Y 474.782,Z 736.686,A -85,B 0,C 180,E1 6924.518,E2 6924.518} C_VEL
LIN {X 0,Y 479.226,Z 688.734,A -85,B 0,C 180,E1 6928.41,E2 6928.41} C_VEL
LIN {X 0,Y 482.582,Z 633.391,A -85,B 0,C 180,E1 6930.626,E2 6930.626} C_VEL
LIN {X 0,Y 480.136,Z 616.815,A -85,B 0,C 180,E1 6931.167,E2 6931.167} C_VEL
LIN {X 0,Y 467.05,Z 586.94,A -85,B 0,C 180,E1 6933.027,E2 6933.027} C_VEL
LIN {X 0,Y 466.735,Z 586.94,A -85,B 0,C 180,E1 6942.202,E2 6942.202} C_VEL
LIN {X 0,Y 466.518,Z 586.94,A -85,B 0,C 180,E1 6951.98,E2 6951.98} C_VEL
LIN {X 0,Y 466.115,Z 586.94,A -85,B 0,C 180,E1 6962.493,E2 6962.493} C_VEL
LIN {X 0,Y 465.998,Z 586.94,A -85,B 0,C 180,E1 6972.858,E2 6972.858} C_VEL
LIN {X 0,Y 465.961,Z 586.94,A -85,B 0,C 180,E1 6982.932,E2 6982.932} C_VEL
LIN {X 0,Y 466.21,Z 586.94,A -85,B 0,C 180,E1 6991.809,E2 6991.809} C_VEL
LIN {X 0,Y 466.788,Z 586.94,A -85,B 0,C 180,E1 7003.547,E2 7003.547} C_VEL
LIN {X 0,Y 467.099,Z 586.94,A -85,B 0,C 180,E1 7013.438,E2 7013.438} C_VEL
LIN {X 0,Y 467.139,Z 586.94,A -85,B 0,C 180,E1 7022.756,E2 7022.756} C_VEL
LIN {X 0,Y 466.697,Z 586.94,A -85,B 0,C 180,E1 7032.16,E2 7032.16} C_VEL
LIN {X 0,Y 466.458,Z 586.94,A -85,B 0,C 180,E1 7041.998,E2 7041.998} C_VEL
LIN {X 0,Y 466.044,Z 586.94,A -85,B 0,C 180,E1 7052.441,E2 7052.441} C_VEL
LIN {X 0,Y 465.95,Z 586.94,A -85,B 0,C 180,E1 7062.878,E2 7062.878} C_VEL
LIN {X 0,Y 466.222,Z 588.478,A -85,B 0,C 180,E1 7064.593,E2 7064.593} C_VEL
LIN {X 0,Y 494.558,Z 642.018,A -85,B 0,C 180,E1 7068.101,E2 7068.101} C_VEL
LIN {X 0,Y 491.588,Z 711.812,A -85,B 0,C 180,E1 7069.882,E2 7069.882} C_VEL
LIN {X 0,Y 482.25,Z 744.899,A -85,B 0,C 180,E1 7070.929,E2 7070.929} C_VEL
LIN {X 0,Y 475.129,Z 806.703,A -85,B 0,C 180,E1 7075.271,E2 7075.271} C_VEL
LIN {X 0,Y 468.617,Z 854.202,A -85,B 0,C 180,E1 7080.564,E2 7080.564} C_VEL
LIN {X 0,Y 462.668,Z 896.926,A -85,B 0,C 180,E1 7087.839,E2 7087.839} C_VEL
LIN {X 0,Y 459.833,Z 925.999,A -85,B 0,C 180,E1 7095.669,E2 7095.669} C_VEL
LIN {X 0,Y 458.977,Z 941.682,A -85,B 0,C 180,E1 7103.354,E2 7103.354} C_VEL
LIN {X 0,Y 458.947,Z 945.837,A -85,B 0,C 180,E1 7110.946,E2 7110.946} C_VEL
LIN {X 0,Y 459.479,Z 938.887,A -85,B 0,C 180,E1 7118.546,E2 7118.546} C_VEL
LIN {X 0,Y 460.745,Z 917.973,A -85,B 0,C 180,E1 7126.919,E2 7126.919} C_VEL
LIN {X 0,Y 464.733,Z 881.732,A -85,B 0,C 180,E1 7135.118,E2 7135.118} C_VEL
LIN {X 0,Y 471.751,Z 833.454,A -85,B 0,C 180,E1 7142.056,E2 7142.056} C_VEL
LIN {X 0,Y 478.804,Z 775.855,A -85,B 0,C 180,E1 7147.124,E2 7147.124} C_VEL
LIN {X 0,Y 484.72,Z 709.378,A -85,B 0,C 180,E1 7150.673,E2 7150.673} C_VEL
LIN {X 0,Y 486.434,Z 641.547,A -85,B 0,C 180,E1 7152.461,E2 7152.461} C_VEL
LIN {X 0,Y 458.036,Z 586.94,A -85,B 0,C 180,E1 7156.176,E2 7156.176} C_VEL
LIN {X 0,Y 457.986,Z 586.94,A -85,B 0,C 180,E1 7166.916,E2 7166.916} C_VEL
LIN {X 0,Y 458.036,Z 586.94,A -85,B 0,C 180,E1 7175.656,E2 7175.656} C_VEL
LIN {X 0,Y 458.404,Z 586.94,A -85,B 0,C 180,E1 7185.667,E2 7185.667} C_VEL
LIN {X 0,Y 458.779,Z 586.94,A -85,B 0,C 180,E1 7195.295,E2 7195.295} C_VEL
LIN {X 0,Y 458.81,Z 586.94,A -85,B 0,C 180,E1 7202.879,E2 7202.879} C_VEL
LIN {X 0,Y 458.771,Z 586.94,A -85,B 0,C 180,E1 7212.635,E2 7212.635} C_VEL
LIN {X 0,Y 458.378,Z 586.94,A -85,B 0,C 180,E1 7222.408,E2 7222.408} C_VEL
LIN {X 0,Y 458.137,Z 586.94,A -85,B 0,C 180,E1 7233.158,E2 7233.158} C_VEL
LIN {X 0,Y 458.594,Z 589.389,A -85,B 0,C 180,E1 7233.871,E2 7233.871} C_VEL
LIN {X 0,Y 477.197,Z 630.005,A -85,B 0,C 180,E1 7236.447,E2 7236.447} C_VEL
LIN {X 0,Y 473.682,Z 685.588,A -85,B 0,C 180,E1 7238.588,E2 7238.588} C_VEL
LIN {X 0,Y 468.532,Z 734.302,A -85,B 0,C 180,E1 7242.405,E2 7242.405} C_VEL
LIN {X 0,Y 463.644,Z 774.03,A -85,B 0,C 180,E1 7247.859,E2 7247.859} C_VEL
LIN {X 0,Y 460.684,Z 800.255,A -85,B 0,C 180,E1 7254.298,E2 7254.298} C_VEL
LIN {X 0,Y 459.622,Z 812.254,A -85,B 0,C 180,E1 7261.071,E2 7261.071} C_VEL
LIN {X 0,Y 459.95,Z 811.216,A -85,B 0,C 180,E1 7267.703,E2 7267.703} C_VEL
LIN {X 0,Y 461.332,Z 795.937,A -85,B 0,C 180,E1 7274.744,E2 7274.744} C_VEL
LIN {X 0,Y 464.321,Z 766.587,A -85,B 0,C 180,E1 7281.07,E2 7281.07} C_VEL
LIN {X 0,Y 468.777,Z 726.235,A -85,B 0,C 180,E1 7286.056,E2 7286.056} C_VEL
LIN {X 0,Y 473.177,Z 677.028,A -85,B 0,C 180,E1 7289.56,E2 7289.56} C_VEL
LIN {X 0,Y 474.652,Z 622.148,A -85,B 0,C 180,E1 7291.495,E2 7291.495} C_VEL
LIN {X 0,Y 458.91,Z 586.94,A -85,B 0,C 180,E1 7293.792,E2 7293.792} C_VEL
LIN {X 0,Y 458.7,Z 586.94,A -85,B 0,C 180,E1 7302.528,E2 7302.528} C_VEL
LIN {X 0,Y 458.495,Z 586.94,A -85,B 0,C 180,E1 7312.373,E2 7312.373} C_VEL
LIN {X 0,Y 458.061,Z 586.94,A -85,B 0,C 180,E1 7323.137,E2 7323.137} C_VEL
LIN {X 0,Y 457.994,Z 586.94,A -85,B 0,C 180,E1 7332.786,E2 7332.786} C_VEL
LIN {X 0,Y 457.868,Z 586.94,A -85,B 0,C 180,E1 7342.154,E2 7342.154} C_VEL
LIN {X 0,Y 458.171,Z 586.94,A -85,B 0,C 180,E1 7351.369,E2 7351.369} C_VEL
LIN {X 0,Y 458.349,Z 586.94,A -85,B 0,C 180,E1 7361.637,E2 7361.637} C_VEL
LIN {X 0,Y 458.779,Z 586.94,A -85,B 0,C 180,E1 7369.486,E2 7369.486} C_VEL
LIN {X 0,Y 459.006,Z 586.94,A -85,B 0,C 180,E1 7379.017,E2 7379.017} C_VEL
LIN {X 0,Y 459.061,Z 586.94,A -85,B 0,C 180,E1 7388.515,E2 7388.515} C_VEL
LIN {X 0,Y 458.44,Z 586.94,A -85,B 0,C 180,E1 7399.367,E2 7399.367} C_VEL
LIN {X 0,Y 458.19,Z 586.94,A -85,B 0,C 180,E1 7408.647,E2 7408.647} C_VEL
LIN {X 0,Y 457.934,Z 586.94,A -85,B 0,C 180,E1 7418.852,E2 7418.852} C_VEL
